KUKA KRL program: EPS_2_251546_SANMH1A_A_20251029061754.src

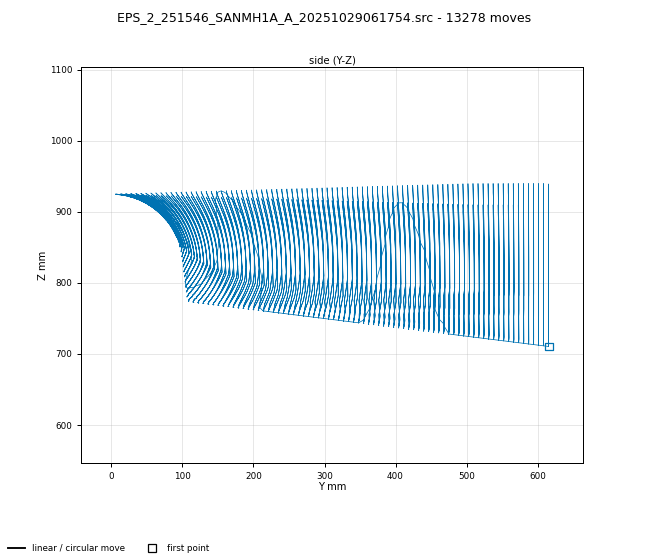
[picture p0: tool path of EPS_2_251546_SANMH1A_A_20251029061754.src, 13278 of 13280 moves have a stored position in this frame; points joined in program order, loops and branches not executed]
&ACCESS RVP
&REL 4
&COMMENT QRS 19112012
&PARAM EDITMASK = *
DEF PART()
EXT BAS (BAS_COMMAND :IN,REAL :IN )
INT I
BAS (#INITMOV,0 )

;KUKA QRS Post kuka4.cps  Date:22-06-2017 !

File_ID=2897

QRS_PRE_INIT()

;Init var - Until changes are made in qrs_pre_init
Outlet_Square_prg=0
Inlet_1_Square_prg=0
Inlet_2_Square_prg=0
Inlet_3_Square_prg=0
Inlet_4_Square_prg=0
Inlet_5_Square_prg=0

Outlet_1={X 0.000, Y 508.730, Z 865.000, B 0.000, E1 0.000 }
Inlet_1={X 0.000, Y 510.870, Z 835.000, B 0.000, E1 180.000 }
Outlet_1_type=150
Inlet_1_type=150
;QRS#1=Sidecore dimensions
;QRS#2=150-6" PVC SDR 28
;QRS#3=150-6" PVC SDR 28
;QRS#4=
;QRS#5=
;QRS#6=
;QRS#7=
;QRS#8=
;QRS#9=10-06 PSX
;QRS#10=10-06 PSX
;QRS#11=
;QRS#12=
;QRS#13=
;QRS#14=
;QRS#15=
;QRS#16=1220x127x1219 4'
;QRS#17=EPS Height
;QRS#18=940
;QRS#19=*
;QRS#20= UPDATED VERSION 22-06-2017
;QRS#21=*
Outlet_Square=070
Inlet_1_Square=070
Inlet_2_Square=0
Inlet_3_Square=0
Inlet_4_Square=0
Inlet_5_Square=0
Mill_Square=1
Outlet_Square_Prg=203
Inlet_1_Square_prg=203

QRS_INIT()

$ADVANCE=5

; T1
PTP {E1 173.424,E2 173.424}
PTP {X 0,Y 615.486,A -85,B 0,C 180,E1 173.424,E2 173.424,E3 0,E4 0,E5 0,E6 0}
QRS_SPEED_INIT()
LIN {X 0,Y 615.486,Z 710.513,A -85,B 0,C 180,E1 173.424,E2 173.424,E3 0,E4 0,E5 0,E6 0} C_VEL
LIN {X 0,Y 615.473,Z 710.502,A -85,B 0,C 180,E1 170.801,E2 170.801} C_VEL
LIN {X 0,Y 615.49,Z 710.493,A -85,B 0,C 180,E1 168.139,E2 168.139} C_VEL
LIN {X 0,Y 615.483,Z 710.506,A -85,B 0,C 180,E1 165.451,E2 165.451} C_VEL
LIN {X 0,Y 615.472,Z 710.505,A -85,B 0,C 180,E1 162.729,E2 162.729} C_VEL
LIN {X 0,Y 615.49,Z 710.493,A -85,B 0,C 180,E1 159.967,E2 159.967} C_VEL
LIN {X 0,Y 615.484,Z 710.511,A -85,B 0,C 180,E1 157.155,E2 157.155} C_VEL
LIN {X 0,Y 615.465,Z 710.503,A -85,B 0,C 180,E1 154.436,E2 154.436} C_VEL
LIN {X 0,Y 615.471,Z 710.498,A -85,B 0,C 180,E1 152.084,E2 152.084} C_VEL
LIN {X 0,Y 615.478,Z 710.496,A -85,B 0,C 180,E1 149.839,E2 149.839} C_VEL
LIN {X 0,Y 615.499,Z 710.493,A -85,B 0,C 180,E1 147.543,E2 147.543} C_VEL
LIN {X 0,Y 615.495,Z 710.499,A -85,B 0,C 180,E1 145.185,E2 145.185} C_VEL
LIN {X 0,Y 615.489,Z 710.514,A -85,B 0,C 180,E1 142.758,E2 142.758} C_VEL
LIN {X 0,Y 615.461,Z 710.501,A -85,B 0,C 180,E1 139.914,E2 139.914} C_VEL
LIN {X 0,Y 615.469,Z 710.497,A -85,B 0,C 180,E1 137.645,E2 137.645} C_VEL
LIN {X 0,Y 615.495,Z 710.5,A -85,B 0,C 180,E1 134.932,E2 134.932} C_VEL
LIN {X 0,Y 615.48,Z 710.511,A -85,B 0,C 180,E1 132.354,E2 132.354} C_VEL
LIN {X 0,Y 615.455,Z 710.503,A -85,B 0,C 180,E1 129.753,E2 129.753} C_VEL
LIN {X 0,Y 615.495,Z 710.497,A -85,B 0,C 180,E1 126.937,E2 126.937} C_VEL
LIN {X 0,Y 615.467,Z 710.508,A -85,B 0,C 180,E1 124.023,E2 124.023} C_VEL
LIN {X 0,Y 615.452,Z 710.505,A -85,B 0,C 180,E1 121.688,E2 121.688} C_VEL
LIN {X 0,Y 615.449,Z 710.503,A -85,B 0,C 180,E1 119.408,E2 119.408} C_VEL
LIN {X 0,Y 615.465,Z 710.499,A -85,B 0,C 180,E1 117.041,E2 117.041} C_VEL
LIN {X 0,Y 615.483,Z 710.511,A -85,B 0,C 180,E1 114.007,E2 114.007} C_VEL
LIN {X 0,Y 615.447,Z 710.505,A -85,B 0,C 180,E1 111.433,E2 111.433} C_VEL
LIN {X 0,Y 615.445,Z 710.505,A -85,B 0,C 180,E1 109.339,E2 109.339} C_VEL
LIN {X 0,Y 615.497,Z 710.635,A -85,B 0,C 180,E1 107.957,E2 107.957} C_VEL
LIN {X 0,Y 615.475,Z 724.409,A -85,B 0,C 180,E1 105.226,E2 105.226} C_VEL
LIN {X 0,Y 615.489,Z 740.007,A -85,B 0,C 180,E1 102.195,E2 102.195} C_VEL
LIN {X 0,Y 615.485,Z 751.04,A -85,B 0,C 180,E1 100.111,E2 100.111} C_VEL
LIN {X 0,Y 615.481,Z 752.153,A -85,B 0,C 180,E1 100.049,E2 100.049} C_VEL
LIN {X 0,Y 615.495,Z 826.708,A -85,B 0,C 180,E1 99.157,E2 99.157} C_VEL
LIN {X 0,Y 615.497,Z 834.892,A -85,B 0,C 180,E1 98.992,E2 98.992} C_VEL
LIN {X 0,Y 615.497,Z 843.45,A -85,B 0,C 180,E1 98.743,E2 98.743} C_VEL
LIN {X 0,Y 615.497,Z 851.061,A -85,B 0,C 180,E1 98.454,E2 98.454} C_VEL
LIN {X 0,Y 615.499,Z 859.582,A -85,B 0,C 180,E1 98.041,E2 98.041} C_VEL
LIN {X 0,Y 615.488,Z 867.749,A -85,B 0,C 180,E1 97.546,E2 97.546} C_VEL
LIN {X 0,Y 615.492,Z 874.389,A -85,B 0,C 180,E1 97.058,E2 97.058} C_VEL
LIN {X 0,Y 615.498,Z 880.184,A -85,B 0,C 180,E1 96.557,E2 96.557} C_VEL
LIN {X 0,Y 615.499,Z 886.535,A -85,B 0,C 180,E1 95.898,E2 95.898} C_VEL
LIN {X 0,Y 615.495,Z 892.984,A -85,B 0,C 180,E1 95.077,E2 95.077} C_VEL
LIN {X 0,Y 615.491,Z 898.123,A -85,B 0,C 180,E1 94.256,E2 94.256} C_VEL
LIN {X 0,Y 615.493,Z 902.886,A -85,B 0,C 180,E1 93.273,E2 93.273} C_VEL
LIN {X 0,Y 615.493,Z 905.2,A -85,B 0,C 180,E1 92.618,E2 92.618} C_VEL
LIN {X 0,Y 615.499,Z 906.976,A -85,B 0,C 180,E1 91.963,E2 91.963} C_VEL
LIN {X 0,Y 615.492,Z 908.266,A -85,B 0,C 180,E1 91.309,E2 91.309} C_VEL
LIN {X 0,Y 615.491,Z 909.083,A -85,B 0,C 180,E1 90.654,E2 90.654} C_VEL
LIN {X 0,Y 615.492,Z 909.384,A -85,B 0,C 180,E1 90,E2 90} C_VEL
LIN {X 0,Y 615.492,Z 909.125,A -85,B 0,C 180,E1 89.346,E2 89.346} C_VEL
LIN {X 0,Y 615.494,Z 908.393,A -85,B 0,C 180,E1 88.691,E2 88.691} C_VEL
LIN {X 0,Y 615.499,Z 907.194,A -85,B 0,C 180,E1 88.037,E2 88.037} C_VEL
LIN {X 0,Y 615.49,Z 904.376,A -85,B 0,C 180,E1 87.055,E2 87.055} C_VEL
LIN {X 0,Y 615.491,Z 901.81,A -85,B 0,C 180,E1 86.399,E2 86.399} C_VEL
LIN {X 0,Y 615.495,Z 896.743,A -85,B 0,C 180,E1 85.416,E2 85.416} C_VEL
LIN {X 0,Y 615.496,Z 891.288,A -85,B 0,C 180,E1 84.595,E2 84.595} C_VEL
LIN {X 0,Y 615.499,Z 884.452,A -85,B 0,C 180,E1 83.773,E2 83.773} C_VEL
LIN {X 0,Y 615.497,Z 877.419,A -85,B 0,C 180,E1 83.1,E2 83.1} C_VEL
LIN {X 0,Y 615.485,Z 869.071,A -85,B 0,C 180,E1 82.454,E2 82.454} C_VEL
LIN {X 0,Y 615.499,Z 861.194,A -85,B 0,C 180,E1 81.959,E2 81.959} C_VEL
LIN {X 0,Y 615.497,Z 853.071,A -85,B 0,C 180,E1 81.546,E2 81.546} C_VEL
LIN {X 0,Y 615.497,Z 844.859,A -85,B 0,C 180,E1 81.215,E2 81.215} C_VEL
LIN {X 0,Y 615.497,Z 836.834,A -85,B 0,C 180,E1 80.967,E2 80.967} C_VEL
LIN {X 0,Y 615.498,Z 827.153,A -85,B 0,C 180,E1 80.76,E2 80.76} C_VEL
LIN {X 0,Y 615.489,Z 751.762,A -85,B 0,C 180,E1 79.847,E2 79.847} C_VEL
LIN {X 0,Y 615.486,Z 750.478,A -85,B 0,C 180,E1 79.722,E2 79.722} C_VEL
LIN {X 0,Y 615.491,Z 735.264,A -85,B 0,C 180,E1 76.799,E2 76.799} C_VEL
LIN {X 0,Y 615.458,Z 721.41,A -85,B 0,C 180,E1 74.094,E2 74.094} C_VEL
LIN {X 0,Y 615.495,Z 710.569,A -85,B 0,C 180,E1 71.922,E2 71.922} C_VEL
LIN {X 0,Y 615.475,Z 710.5,A -85,B 0,C 180,E1 69.269,E2 69.269} C_VEL
LIN {X 0,Y 615.469,Z 710.5,A -85,B 0,C 180,E1 67.155,E2 67.155} C_VEL
LIN {X 0,Y 615.464,Z 710.5,A -85,B 0,C 180,E1 65.007,E2 65.007} C_VEL
LIN {X 0,Y 615.452,Z 710.502,A -85,B 0,C 180,E1 62.821,E2 62.821} C_VEL
LIN {X 0,Y 615.444,Z 710.503,A -85,B 0,C 180,E1 60.591,E2 60.591} C_VEL
LIN {X 0,Y 615.444,Z 710.506,A -85,B 0,C 180,E1 58.312,E2 58.312} C_VEL
LIN {X 0,Y 615.457,Z 710.508,A -85,B 0,C 180,E1 55.976,E2 55.976} C_VEL
LIN {X 0,Y 615.495,Z 710.498,A -85,B 0,C 180,E1 53.063,E2 53.063} C_VEL
LIN {X 0,Y 615.451,Z 710.503,A -85,B 0,C 180,E1 50.247,E2 50.247} C_VEL
LIN {X 0,Y 615.474,Z 710.51,A -85,B 0,C 180,E1 47.646,E2 47.646} C_VEL
LIN {X 0,Y 615.497,Z 710.498,A -85,B 0,C 180,E1 44.932,E2 44.932} C_VEL
LIN {X 0,Y 615.467,Z 710.498,A -85,B 0,C 180,E1 42.355,E2 42.355} C_VEL
LIN {X 0,Y 615.459,Z 710.506,A -85,B 0,C 180,E1 39.752,E2 39.752} C_VEL
LIN {X 0,Y 615.492,Z 710.504,A -85,B 0,C 180,E1 36.937,E2 36.937} C_VEL
LIN {X 0,Y 615.464,Z 710.499,A -85,B 0,C 180,E1 34.024,E2 34.024} C_VEL
LIN {X 0,Y 615.46,Z 710.503,A -85,B 0,C 180,E1 31.687,E2 31.687} C_VEL
LIN {X 0,Y 615.469,Z 710.507,A -85,B 0,C 180,E1 29.407,E2 29.407} C_VEL
LIN {X 0,Y 615.494,Z 710.496,A -85,B 0,C 180,E1 26.444,E2 26.444} C_VEL
LIN {X 0,Y 615.484,Z 710.494,A -85,B 0,C 180,E1 24.007,E2 24.007} C_VEL
LIN {X 0,Y 615.465,Z 710.503,A -85,B 0,C 180,E1 21.433,E2 21.433} C_VEL
LIN {X 0,Y 615.489,Z 710.506,A -85,B 0,C 180,E1 18.605,E2 18.605} C_VEL
LIN {X 0,Y 615.488,Z 710.494,A -85,B 0,C 180,E1 15.905,E2 15.905} C_VEL
LIN {X 0,Y 615.47,Z 710.504,A -85,B 0,C 180,E1 13.202,E2 13.202} C_VEL
LIN {X 0,Y 615.486,Z 710.51,A -85,B 0,C 180,E1 10.527,E2 10.527} C_VEL
LIN {X 0,Y 615.495,Z 710.493,A -85,B 0,C 180,E1 7.876,E2 7.876} C_VEL
LIN {X 0,Y 615.474,Z 710.499,A -85,B 0,C 180,E1 5.241,E2 5.241} C_VEL
LIN {X 0,Y 615.491,Z 710.511,A -85,B 0,C 180,E1 2.618,E2 2.618} C_VEL
LIN {X 0,Y 615.486,Z 710.5,A -85,B 0,C 180,E1 0,E2 0} C_VEL
LIN {X 0,Y 615.495,Z 710.492,A -85,B 0,C 180,E1 -2.618,E2 -2.618} C_VEL
LIN {X 0,Y 615.477,Z 710.504,A -85,B 0,C 180,E1 -5.241,E2 -5.241} C_VEL
LIN {X 0,Y 615.485,Z 710.508,A -85,B 0,C 180,E1 -7.876,E2 -7.876} C_VEL
LIN {X 0,Y 615.492,Z 710.493,A -85,B 0,C 180,E1 -10.527,E2 -10.527} C_VEL
LIN {X 0,Y 615.481,Z 710.499,A -85,B 0,C 180,E1 -13.201,E2 -13.201} C_VEL
LIN {X 0,Y 615.483,Z 710.514,A -85,B 0,C 180,E1 -15.905,E2 -15.905} C_VEL
LIN {X 0,Y 615.492,Z 710.494,A -85,B 0,C 180,E1 -18.646,E2 -18.646} C_VEL
LIN {X 0,Y 615.483,Z 710.5,A -85,B 0,C 180,E1 -21.432,E2 -21.432} C_VEL
LIN {X 0,Y 615.485,Z 710.506,A -85,B 0,C 180,E1 -24.272,E2 -24.272} C_VEL
LIN {X 0,Y 615.489,Z 710.493,A -85,B 0,C 180,E1 -27.177,E2 -27.177} C_VEL
LIN {X 0,Y 615.485,Z 710.504,A -85,B 0,C 180,E1 -29.794,E2 -29.794} C_VEL
LIN {X 0,Y 615.479,Z 710.506,A -85,B 0,C 180,E1 -32.458,E2 -32.458} C_VEL
LIN {X 0,Y 615.497,Z 710.495,A -85,B 0,C 180,E1 -34.814,E2 -34.814} C_VEL
LIN {X 0,Y 615.488,Z 710.493,A -85,B 0,C 180,E1 -37.242,E2 -37.242} C_VEL
LIN {X 0,Y 615.489,Z 710.506,A -85,B 0,C 180,E1 -40.089,E2 -40.089} C_VEL
LIN {X 0,Y 615.498,Z 710.513,A -85,B 0,C 180,E1 -42.352,E2 -42.352} C_VEL
LIN {X 0,Y 615.495,Z 710.494,A -85,B 0,C 180,E1 -45.068,E2 -45.068} C_VEL
LIN {X 0,Y 615.495,Z 710.496,A -85,B 0,C 180,E1 -47.919,E2 -47.919} C_VEL
LIN {X 0,Y 615.49,Z 710.505,A -85,B 0,C 180,E1 -50.25,E2 -50.25} C_VEL
LIN {X 0,Y 615.48,Z 710.501,A -85,B 0,C 180,E1 -53.064,E2 -53.064} C_VEL
LIN {X 0,Y 615.49,Z 710.495,A -85,B 0,C 180,E1 -55.299,E2 -55.299} C_VEL
LIN {X 0,Y 615.484,Z 710.494,A -85,B 0,C 180,E1 -57.67,E2 -57.67} C_VEL
LIN {X 0,Y 615.489,Z 710.51,A -85,B 0,C 180,E1 -60.594,E2 -60.594} C_VEL
LIN {X 0,Y 615.475,Z 710.511,A -85,B 0,C 180,E1 -62.957,E2 -62.957} C_VEL
LIN {X 0,Y 615.484,Z 710.494,A -85,B 0,C 180,E1 -65.728,E2 -65.728} C_VEL
LIN {X 0,Y 615.495,Z 710.502,A -85,B 0,C 180,E1 -68.568,E2 -68.568} C_VEL
LIN {X 0,Y 615.498,Z 710.672,A -85,B 0,C 180,E1 -68.963,E2 -68.963} C_VEL
LIN {X 0,Y 615.491,Z 726.63,A -85,B 0,C 180,E1 -71.557,E2 -71.557} C_VEL
LIN {X 0,Y 615.496,Z 744.77,A -85,B 0,C 180,E1 -74.435,E2 -74.435} C_VEL
LIN {X 0,Y 615.478,Z 763.08,A -85,B 0,C 180,E1 -77.302,E2 -77.302} C_VEL
LIN {X 0,Y 615.493,Z 779.482,A -85,B 0,C 180,E1 -79.826,E2 -79.826} C_VEL
LIN {X 0,Y 615.491,Z 780.6,A -85,B 0,C 180,E1 -79.889,E2 -79.889} C_VEL
LIN {X 0,Y 615.499,Z 856.93,A -85,B 0,C 180,E1 -80.801,E2 -80.801} C_VEL
LIN {X 0,Y 615.497,Z 866.69,A -85,B 0,C 180,E1 -81.008,E2 -81.008} C_VEL
LIN {X 0,Y 615.498,Z 877.15,A -85,B 0,C 180,E1 -81.339,E2 -81.339} C_VEL
LIN {X 0,Y 615.497,Z 887.426,A -85,B 0,C 180,E1 -81.794,E2 -81.794} C_VEL
LIN {X 0,Y 615.491,Z 897.198,A -85,B 0,C 180,E1 -82.372,E2 -82.372} C_VEL
LIN {X 0,Y 615.498,Z 904.934,A -85,B 0,C 180,E1 -82.942,E2 -82.942} C_VEL
LIN {X 0,Y 615.498,Z 910.646,A -85,B 0,C 180,E1 -83.443,E2 -83.443} C_VEL
LIN {X 0,Y 615.499,Z 916.921,A -85,B 0,C 180,E1 -84.102,E2 -84.102} C_VEL
LIN {X 0,Y 615.496,Z 922.135,A -85,B 0,C 180,E1 -84.759,E2 -84.759} C_VEL
LIN {X 0,Y 615.495,Z 926.482,A -85,B 0,C 180,E1 -85.416,E2 -85.416} C_VEL
LIN {X 0,Y 615.492,Z 931.603,A -85,B 0,C 180,E1 -86.399,E2 -86.399} C_VEL
LIN {X 0,Y 615.488,Z 934.221,A -85,B 0,C 180,E1 -87.055,E2 -87.055} C_VEL
LIN {X 0,Y 615.495,Z 937.086,A -85,B 0,C 180,E1 -88.037,E2 -88.037} C_VEL
LIN {X 0,Y 615.494,Z 938.33,A -85,B 0,C 180,E1 -88.691,E2 -88.691} C_VEL
LIN {X 0,Y 615.493,Z 939.104,A -85,B 0,C 180,E1 -89.346,E2 -89.346} C_VEL
LIN {X 0,Y 615.491,Z 939.389,A -85,B 0,C 180,E1 -90,E2 -90} C_VEL
LIN {X 0,Y 615.493,Z 939.104,A -85,B 0,C 180,E1 -90.654,E2 -90.654} C_VEL
LIN {X 0,Y 615.494,Z 938.33,A -85,B 0,C 180,E1 -91.309,E2 -91.309} C_VEL
LIN {X 0,Y 615.495,Z 937.086,A -85,B 0,C 180,E1 -91.963,E2 -91.963} C_VEL
LIN {X 0,Y 615.488,Z 934.221,A -85,B 0,C 180,E1 -92.945,E2 -92.945} C_VEL
LIN {X 0,Y 615.492,Z 931.603,A -85,B 0,C 180,E1 -93.601,E2 -93.601} C_VEL
LIN {X 0,Y 615.495,Z 926.482,A -85,B 0,C 180,E1 -94.584,E2 -94.584} C_VEL
LIN {X 0,Y 615.495,Z 920.968,A -85,B 0,C 180,E1 -95.405,E2 -95.405} C_VEL
LIN {X 0,Y 615.498,Z 914.018,A -85,B 0,C 180,E1 -96.227,E2 -96.227} C_VEL
LIN {X 0,Y 615.497,Z 906.858,A -85,B 0,C 180,E1 -96.901,E2 -96.901} C_VEL
LIN {X 0,Y 615.488,Z 899.621,A -85,B 0,C 180,E1 -97.463,E2 -97.463} C_VEL
LIN {X 0,Y 615.497,Z 891.868,A -85,B 0,C 180,E1 -97.958,E2 -97.958} C_VEL
LIN {X 0,Y 615.498,Z 883.913,A -85,B 0,C 180,E1 -98.371,E2 -98.371} C_VEL
LIN {X 0,Y 615.497,Z 874.754,A -85,B 0,C 180,E1 -98.743,E2 -98.743} C_VEL
LIN {X 0,Y 615.497,Z 866.69,A -85,B 0,C 180,E1 -98.992,E2 -98.992} C_VEL
LIN {X 0,Y 615.499,Z 856.93,A -85,B 0,C 180,E1 -99.199,E2 -99.199} C_VEL
LIN {X 0,Y 615.491,Z 780.6,A -85,B 0,C 180,E1 -100.111,E2 -100.111} C_VEL
LIN {X 0,Y 615.493,Z 779.29,A -85,B 0,C 180,E1 -100.194,E2 -100.194} C_VEL
LIN {X 0,Y 615.479,Z 762.006,A -85,B 0,C 180,E1 -102.866,E2 -102.866} C_VEL
LIN {X 0,Y 615.497,Z 743.691,A -85,B 0,C 180,E1 -105.735,E2 -105.735} C_VEL
LIN {X 0,Y 615.49,Z 725.613,A -85,B 0,C 180,E1 -108.606,E2 -108.606} C_VEL
LIN {X 0,Y 615.498,Z 710.672,A -85,B 0,C 180,E1 -111.037,E2 -111.037} C_VEL
LIN {X 0,Y 615.491,Z 710.501,A -85,B 0,C 180,E1 -113.556,E2 -113.556} C_VEL
LIN {X 0,Y 615.486,Z 710.495,A -85,B 0,C 180,E1 -116.444,E2 -116.444} C_VEL
LIN {X 0,Y 615.485,Z 710.497,A -85,B 0,C 180,E1 -118.658,E2 -118.658} C_VEL
LIN {X 0,Y 615.485,Z 710.507,A -85,B 0,C 180,E1 -121.086,E2 -121.086} C_VEL
LIN {X 0,Y 615.492,Z 710.495,A -85,B 0,C 180,E1 -124.022,E2 -124.022} C_VEL
LIN {X 0,Y 615.484,Z 710.494,A -85,B 0,C 180,E1 -126.425,E2 -126.425} C_VEL
LIN {X 0,Y 615.481,Z 710.503,A -85,B 0,C 180,E1 -129.061,E2 -129.061} C_VEL
LIN {X 0,Y 615.49,Z 710.513,A -85,B 0,C 180,E1 -131.474,E2 -131.474} C_VEL
LIN {X 0,Y 615.496,Z 710.496,A -85,B 0,C 180,E1 -134.149,E2 -134.149} C_VEL
LIN {X 0,Y 615.492,Z 710.495,A -85,B 0,C 180,E1 -136.952,E2 -136.952} C_VEL
LIN {X 0,Y 615.482,Z 710.506,A -85,B 0,C 180,E1 -139.393,E2 -139.393} C_VEL
LIN {X 0,Y 615.489,Z 710.506,A -85,B 0,C 180,E1 -141.988,E2 -141.988} C_VEL
LIN {X 0,Y 615.493,Z 710.496,A -85,B 0,C 180,E1 -144.385,E2 -144.385} C_VEL
LIN {X 0,Y 615.491,Z 710.493,A -85,B 0,C 180,E1 -146.764,E2 -146.764} C_VEL
LIN {X 0,Y 615.49,Z 710.494,A -85,B 0,C 180,E1 -149.08,E2 -149.08} C_VEL
LIN {X 0,Y 615.478,Z 710.504,A -85,B 0,C 180,E1 -151.552,E2 -151.552} C_VEL
LIN {X 0,Y 615.482,Z 710.506,A -85,B 0,C 180,E1 -154.284,E2 -154.284} C_VEL
LIN {X 0,Y 615.49,Z 710.493,A -85,B 0,C 180,E1 -157.156,E2 -157.156} C_VEL
LIN {X 0,Y 615.482,Z 710.511,A -85,B 0,C 180,E1 -159.967,E2 -159.967} C_VEL
LIN {X 0,Y 615.484,Z 710.498,A -85,B 0,C 180,E1 -162.729,E2 -162.729} C_VEL
LIN {X 0,Y 615.492,Z 710.493,A -85,B 0,C 180,E1 -165.451,E2 -165.451} C_VEL
LIN {X 0,Y 615.484,Z 710.511,A -85,B 0,C 180,E1 -168.139,E2 -168.139} C_VEL
LIN {X 0,Y 615.48,Z 710.501,A -85,B 0,C 180,E1 -170.801,E2 -170.801} C_VEL
LIN {X 0,Y 615.492,Z 710.492,A -85,B 0,C 180,E1 -173.443,E2 -173.443} C_VEL
LIN {X 0,Y 615.49,Z 710.502,A -85,B 0,C 180,E1 -176.072,E2 -176.072} C_VEL
LIN {X 0,Y 615.485,Z 710.508,A -85,B 0,C 180,E1 -178.691,E2 -178.691} C_VEL
LIN {X 0,Y 615.483,Z 710.496,A -85,B 0,C 180,E1 -181.309,E2 -181.309} C_VEL
LIN {X 0,Y 615.495,Z 710.494,A -85,B 0,C 180,E1 -183.929,E2 -183.929} C_VEL
LIN {X 0,Y 615.486,Z 710.513,A -85,B 0,C 180,E1 -186.576,E2 -186.576} C_VEL
LIN {X 0,Y 614.801,Z 710.649,A -85,B 0,C 180,E1 -187.122,E2 -187.122} C_VEL
LIN {X 0,Y 611.958,Z 711.063,A -85,B 0,C 180,E1 -188.008,E2 -188.008} C_VEL
LIN {X 0,Y 609.568,Z 711.374,A -85,B 0,C 180,E1 -188.721,E2 -188.721} C_VEL
LIN {X 0,Y 608.541,Z 711.491,A -85,B 0,C 180,E1 -189.27,E2 -189.27} C_VEL
LIN {X 0,Y 608.455,Z 711.499,A -85,B 0,C 180,E1 -189.456,E2 -189.456} C_VEL
LIN {X 0,Y 608.465,Z 711.498,A -85,B 0,C 180,E1 -192,E2 -192} C_VEL
LIN {X 0,Y 608.47,Z 711.507,A -85,B 0,C 180,E1 -194.721,E2 -194.721} C_VEL
LIN {X 0,Y 608.446,Z 711.501,A -85,B 0,C 180,E1 -197.477,E2 -197.477} C_VEL
LIN {X 0,Y 608.468,Z 711.498,A -85,B 0,C 180,E1 -200.274,E2 -200.274} C_VEL
LIN {X 0,Y 608.443,Z 711.509,A -85,B 0,C 180,E1 -203.124,E2 -203.124} C_VEL
LIN {X 0,Y 608.455,Z 711.5,A -85,B 0,C 180,E1 -205.717,E2 -205.717} C_VEL
LIN {X 0,Y 608.453,Z 711.499,A -85,B 0,C 180,E1 -208.267,E2 -208.267} C_VEL
LIN {X 0,Y 608.468,Z 711.499,A -85,B 0,C 180,E1 -210.545,E2 -210.545} C_VEL
LIN {X 0,Y 608.461,Z 711.504,A -85,B 0,C 180,E1 -212.879,E2 -212.879} C_VEL
LIN {X 0,Y 608.438,Z 711.512,A -85,B 0,C 180,E1 -215.278,E2 -215.278} C_VEL
LIN {X 0,Y 608.456,Z 711.502,A -85,B 0,C 180,E1 -217.747,E2 -217.747} C_VEL
LIN {X 0,Y 608.439,Z 711.5,A -85,B 0,C 180,E1 -220.327,E2 -220.327} C_VEL
LIN {X 0,Y 608.48,Z 711.505,A -85,B 0,C 180,E1 -223.31,E2 -223.31} C_VEL
LIN {X 0,Y 608.451,Z 711.5,A -85,B 0,C 180,E1 -226.129,E2 -226.129} C_VEL
LIN {X 0,Y 608.455,Z 711.5,A -85,B 0,C 180,E1 -228.823,E2 -228.823} C_VEL
LIN {X 0,Y 608.454,Z 711.506,A -85,B 0,C 180,E1 -231.761,E2 -231.761} C_VEL
LIN {X 0,Y 608.439,Z 711.506,A -85,B 0,C 180,E1 -233.956,E2 -233.956} C_VEL
LIN {X 0,Y 608.444,Z 711.501,A -85,B 0,C 180,E1 -236.328,E2 -236.328} C_VEL
LIN {X 0,Y 608.442,Z 711.5,A -85,B 0,C 180,E1 -238.733,E2 -238.733} C_VEL
LIN {X 0,Y 608.481,Z 711.5,A -85,B 0,C 180,E1 -241.379,E2 -241.379} C_VEL
LIN {X 0,Y 608.445,Z 711.503,A -85,B 0,C 180,E1 -244.285,E2 -244.285} C_VEL
LIN {X 0,Y 608.429,Z 711.502,A -85,B 0,C 180,E1 -246.875,E2 -246.875} C_VEL
LIN {X 0,Y 608.465,Z 711.505,A -85,B 0,C 180,E1 -249.726,E2 -249.726} C_VEL
LIN {X 0,Y 608.493,Z 711.606,A -85,B 0,C 180,E1 -252.004,E2 -252.004} C_VEL
LIN {X 0,Y 608.457,Z 724.582,A -85,B 0,C 180,E1 -254.594,E2 -254.594} C_VEL
LIN {X 0,Y 608.458,Z 738.509,A -85,B 0,C 180,E1 -257.323,E2 -257.323} C_VEL
LIN {X 0,Y 608.466,Z 751.478,A -85,B 0,C 180,E1 -259.792,E2 -259.792} C_VEL
LIN {X 0,Y 608.516,Z 753.832,A -85,B 0,C 180,E1 -259.856,E2 -259.856} C_VEL
LIN {X 0,Y 608.508,Z 827.252,A -85,B 0,C 180,E1 -260.737,E2 -260.737} C_VEL
LIN {X 0,Y 608.512,Z 836.951,A -85,B 0,C 180,E1 -260.946,E2 -260.946} C_VEL
LIN {X 0,Y 608.499,Z 848.538,A -85,B 0,C 180,E1 -261.323,E2 -261.323} C_VEL
LIN {X 0,Y 608.479,Z 858.432,A -85,B 0,C 180,E1 -261.782,E2 -261.782} C_VEL
LIN {X 0,Y 608.471,Z 866.885,A -85,B 0,C 180,E1 -262.283,E2 -262.283} C_VEL
LIN {X 0,Y 608.46,Z 874.854,A -85,B 0,C 180,E1 -262.867,E2 -262.867} C_VEL
LIN {X 0,Y 608.467,Z 881.903,A -85,B 0,C 180,E1 -263.496,E2 -263.496} C_VEL
LIN {X 0,Y 608.458,Z 888.396,A -85,B 0,C 180,E1 -264.199,E2 -264.199} C_VEL
LIN {X 0,Y 608.437,Z 894.642,A -85,B 0,C 180,E1 -265.03,E2 -265.03} C_VEL
LIN {X 0,Y 608.432,Z 900.425,A -85,B 0,C 180,E1 -266.026,E2 -266.026} C_VEL
LIN {X 0,Y 608.447,Z 904.63,A -85,B 0,C 180,E1 -267.021,E2 -267.021} C_VEL
LIN {X 0,Y 608.443,Z 907.569,A -85,B 0,C 180,E1 -268.014,E2 -268.014} C_VEL
LIN {X 0,Y 608.445,Z 908.87,A -85,B 0,C 180,E1 -268.676,E2 -268.676} C_VEL
LIN {X 0,Y 608.434,Z 909.692,A -85,B 0,C 180,E1 -269.338,E2 -269.338} C_VEL
LIN {X 0,Y 608.432,Z 909.995,A -85,B 0,C 180,E1 -270,E2 -270} C_VEL
LIN {X 0,Y 608.435,Z 909.735,A -85,B 0,C 180,E1 -270.662,E2 -270.662} C_VEL
LIN {X 0,Y 608.446,Z 908.997,A -85,B 0,C 180,E1 -271.324,E2 -271.324} C_VEL
LIN {X 0,Y 608.444,Z 907.787,A -85,B 0,C 180,E1 -271.986,E2 -271.986} C_VEL
LIN {X 0,Y 608.445,Z 904.941,A -85,B 0,C 180,E1 -272.979,E2 -272.979} C_VEL
LIN {X 0,Y 608.445,Z 902.352,A -85,B 0,C 180,E1 -273.642,E2 -273.642} C_VEL
LIN {X 0,Y 608.445,Z 897.244,A -85,B 0,C 180,E1 -274.638,E2 -274.638} C_VEL
LIN {X 0,Y 608.461,Z 891.748,A -85,B 0,C 180,E1 -275.468,E2 -275.468} C_VEL
LIN {X 0,Y 608.455,Z 884.144,A -85,B 0,C 180,E1 -276.374,E2 -276.374} C_VEL
LIN {X 0,Y 608.463,Z 875.948,A -85,B 0,C 180,E1 -277.133,E2 -277.133} C_VEL
LIN {X 0,Y 608.467,Z 868.198,A -85,B 0,C 180,E1 -277.717,E2 -277.717} C_VEL
LIN {X 0,Y 608.48,Z 860.032,A -85,B 0,C 180,E1 -278.218,E2 -278.218} C_VEL
LIN {X 0,Y 608.484,Z 849.674,A -85,B 0,C 180,E1 -278.719,E2 -278.719} C_VEL
LIN {X 0,Y 608.51,Z 838.029,A -85,B 0,C 180,E1 -279.117,E2 -279.117} C_VEL
LIN {X 0,Y 608.517,Z 827.635,A -85,B 0,C 180,E1 -279.347,E2 -279.347} C_VEL
LIN {X 0,Y 608.509,Z 781.173,A -85,B 0,C 180,E1 -279.913,E2 -279.913} C_VEL
LIN {X 0,Y 608.484,Z 751.922,A -85,B 0,C 180,E1 -280.271,E2 -280.271} C_VEL
LIN {X 0,Y 608.457,Z 750.745,A -85,B 0,C 180,E1 -280.398,E2 -280.398} C_VEL
LIN {X 0,Y 608.463,Z 735.488,A -85,B 0,C 180,E1 -283.356,E2 -283.356} C_VEL
LIN {X 0,Y 608.452,Z 721.556,A -85,B 0,C 180,E1 -286.094,E2 -286.094} C_VEL
LIN {X 0,Y 608.471,Z 711.572,A -85,B 0,C 180,E1 -288.106,E2 -288.106} C_VEL
LIN {X 0,Y 608.438,Z 711.501,A -85,B 0,C 180,E1 -290.982,E2 -290.982} C_VEL
LIN {X 0,Y 608.425,Z 711.503,A -85,B 0,C 180,E1 -293.125,E2 -293.125} C_VEL
LIN {X 0,Y 608.439,Z 711.503,A -85,B 0,C 180,E1 -295.714,E2 -295.714} C_VEL
LIN {X 0,Y 608.482,Z 711.501,A -85,B 0,C 180,E1 -298.621,E2 -298.621} C_VEL
LIN {X 0,Y 608.437,Z 711.501,A -85,B 0,C 180,E1 -301.318,E2 -301.318} C_VEL
LIN {X 0,Y 608.425,Z 711.504,A -85,B 0,C 180,E1 -303.728,E2 -303.728} C_VEL
LIN {X 0,Y 608.439,Z 711.506,A -85,B 0,C 180,E1 -306.093,E2 -306.093} C_VEL
LIN {X 0,Y 608.467,Z 711.507,A -85,B 0,C 180,E1 -308.588,E2 -308.588} C_VEL
LIN {X 0,Y 608.452,Z 711.5,A -85,B 0,C 180,E1 -311.341,E2 -311.341} C_VEL
LIN {X 0,Y 608.446,Z 711.501,A -85,B 0,C 180,E1 -313.872,E2 -313.872} C_VEL
LIN {X 0,Y 608.48,Z 711.506,A -85,B 0,C 180,E1 -316.69,E2 -316.69} C_VEL
LIN {X 0,Y 608.454,Z 711.499,A -85,B 0,C 180,E1 -319.697,E2 -319.697} C_VEL
LIN {X 0,Y 608.481,Z 711.506,A -85,B 0,C 180,E1 -322.84,E2 -322.84} C_VEL
LIN {X 0,Y 608.469,Z 711.498,A -85,B 0,C 180,E1 -325.531,E2 -325.531} C_VEL
LIN {X 0,Y 608.462,Z 711.498,A -85,B 0,C 180,E1 -327.905,E2 -327.905} C_VEL
LIN {X 0,Y 608.448,Z 711.5,A -85,B 0,C 180,E1 -330.219,E2 -330.219} C_VEL
LIN {X 0,Y 608.479,Z 711.503,A -85,B 0,C 180,E1 -332.793,E2 -332.793} C_VEL
LIN {X 0,Y 608.48,Z 711.496,A -85,B 0,C 180,E1 -335.847,E2 -335.847} C_VEL
LIN {X 0,Y 608.461,Z 711.498,A -85,B 0,C 180,E1 -338.308,E2 -338.308} C_VEL
LIN {X 0,Y 608.454,Z 711.51,A -85,B 0,C 180,E1 -341.13,E2 -341.13} C_VEL
LIN {X 0,Y 608.465,Z 711.498,A -85,B 0,C 180,E1 -343.906,E2 -343.906} C_VEL
LIN {X 0,Y 608.454,Z 711.5,A -85,B 0,C 180,E1 -346.643,E2 -346.643} C_VEL
LIN {X 0,Y 608.463,Z 711.509,A -85,B 0,C 180,E1 -349.35,E2 -349.35} C_VEL
LIN {X 0,Y 608.485,Z 711.496,A -85,B 0,C 180,E1 -352.033,E2 -352.033} C_VEL
LIN {X 0,Y 608.456,Z 711.499,A -85,B 0,C 180,E1 -354.698,E2 -354.698} C_VEL
LIN {X 0,Y 608.482,Z 711.505,A -85,B 0,C 180,E1 -357.352,E2 -357.352} C_VEL
LIN {X 0,Y 608.477,Z 711.499,A -85,B 0,C 180,E1 -360,E2 -360} C_VEL
LIN {X 0,Y 608.484,Z 711.495,A -85,B 0,C 180,E1 -362.648,E2 -362.648} C_VEL
LIN {X 0,Y 608.458,Z 711.504,A -85,B 0,C 180,E1 -365.302,E2 -365.302} C_VEL
LIN {X 0,Y 608.479,Z 711.502,A -85,B 0,C 180,E1 -367.967,E2 -367.967} C_VEL
LIN {X 0,Y 608.472,Z 711.497,A -85,B 0,C 180,E1 -370.956,E2 -370.956} C_VEL
LIN {X 0,Y 608.462,Z 711.501,A -85,B 0,C 180,E1 -373.356,E2 -373.356} C_VEL
LIN {X 0,Y 608.462,Z 711.505,A -85,B 0,C 180,E1 -376.094,E2 -376.094} C_VEL
LIN {X 0,Y 608.459,Z 711.498,A -85,B 0,C 180,E1 -378.869,E2 -378.869} C_VEL
LIN {X 0,Y 608.467,Z 711.503,A -85,B 0,C 180,E1 -381.692,E2 -381.692} C_VEL
LIN {X 0,Y 608.455,Z 711.501,A -85,B 0,C 180,E1 -384.571,E2 -384.571} C_VEL
LIN {X 0,Y 608.483,Z 711.495,A -85,B 0,C 180,E1 -387.208,E2 -387.208} C_VEL
LIN {X 0,Y 608.469,Z 711.505,A -85,B 0,C 180,E1 -389.971,E2 -389.971} C_VEL
LIN {X 0,Y 608.456,Z 711.504,A -85,B 0,C 180,E1 -392.521,E2 -392.521} C_VEL
LIN {X 0,Y 608.452,Z 711.499,A -85,B 0,C 180,E1 -395.277,E2 -395.277} C_VEL
LIN {X 0,Y 608.472,Z 711.499,A -85,B 0,C 180,E1 -397.746,E2 -397.746} C_VEL
LIN {X 0,Y 608.452,Z 711.51,A -85,B 0,C 180,E1 -400.329,E2 -400.329} C_VEL
LIN {X 0,Y 608.46,Z 711.5,A -85,B 0,C 180,E1 -402.959,E2 -402.959} C_VEL
LIN {X 0,Y 608.464,Z 711.499,A -85,B 0,C 180,E1 -405.735,E2 -405.735} C_VEL
LIN {X 0,Y 608.465,Z 711.506,A -85,B 0,C 180,E1 -408.657,E2 -408.657} C_VEL
LIN {X 0,Y 608.472,Z 711.497,A -85,B 0,C 180,E1 -411.412,E2 -411.412} C_VEL
LIN {X 0,Y 608.48,Z 711.497,A -85,B 0,C 180,E1 -413.95,E2 -413.95} C_VEL
LIN {X 0,Y 608.469,Z 711.503,A -85,B 0,C 180,E1 -416.33,E2 -416.33} C_VEL
LIN {X 0,Y 608.479,Z 711.507,A -85,B 0,C 180,E1 -418.727,E2 -418.727} C_VEL
LIN {X 0,Y 608.473,Z 711.498,A -85,B 0,C 180,E1 -421.38,E2 -421.38} C_VEL
LIN {X 0,Y 608.481,Z 711.498,A -85,B 0,C 180,E1 -424.277,E2 -424.277} C_VEL
LIN {X 0,Y 608.45,Z 711.511,A -85,B 0,C 180,E1 -426.876,E2 -426.876} C_VEL
LIN {X 0,Y 608.489,Z 711.683,A -85,B 0,C 180,E1 -428.887,E2 -428.887} C_VEL
LIN {X 0,Y 608.514,Z 726.278,A -85,B 0,C 180,E1 -431.272,E2 -431.272} C_VEL
LIN {X 0,Y 608.503,Z 744.878,A -85,B 0,C 180,E1 -434.251,E2 -434.251} C_VEL
LIN {X 0,Y 608.452,Z 763.263,A -85,B 0,C 180,E1 -437.153,E2 -437.153} C_VEL
LIN {X 0,Y 608.47,Z 779.912,A -85,B 0,C 180,E1 -439.729,E2 -439.729} C_VEL
LIN {X 0,Y 608.52,Z 782.297,A -85,B 0,C 180,E1 -439.793,E2 -439.793} C_VEL
LIN {X 0,Y 608.504,Z 856.143,A -85,B 0,C 180,E1 -440.674,E2 -440.674} C_VEL
LIN {X 0,Y 608.496,Z 865.413,A -85,B 0,C 180,E1 -440.862,E2 -440.862} C_VEL
LIN {X 0,Y 608.489,Z 873.887,A -85,B 0,C 180,E1 -441.113,E2 -441.113} C_VEL
LIN {X 0,Y 608.501,Z 882.387,A -85,B 0,C 180,E1 -441.448,E2 -441.448} C_VEL
LIN {X 0,Y 608.497,Z 890.718,A -85,B 0,C 180,E1 -441.866,E2 -441.866} C_VEL
LIN {X 0,Y 608.469,Z 898.759,A -85,B 0,C 180,E1 -442.367,E2 -442.367} C_VEL
LIN {X 0,Y 608.484,Z 906.414,A -85,B 0,C 180,E1 -442.951,E2 -442.951} C_VEL
LIN {X 0,Y 608.452,Z 914.437,A -85,B 0,C 180,E1 -443.7,E2 -443.7} C_VEL
LIN {X 0,Y 608.46,Z 921.43,A -85,B 0,C 180,E1 -444.532,E2 -444.532} C_VEL
LIN {X 0,Y 608.431,Z 926.985,A -85,B 0,C 180,E1 -445.362,E2 -445.362} C_VEL
LIN {X 0,Y 608.446,Z 932.146,A -85,B 0,C 180,E1 -446.358,E2 -446.358} C_VEL
LIN {X 0,Y 608.444,Z 934.786,A -85,B 0,C 180,E1 -447.021,E2 -447.021} C_VEL
LIN {X 0,Y 608.44,Z 937.678,A -85,B 0,C 180,E1 -448.014,E2 -448.014} C_VEL
LIN {X 0,Y 608.446,Z 938.934,A -85,B 0,C 180,E1 -448.676,E2 -448.676} C_VEL
LIN {X 0,Y 608.436,Z 939.714,A -85,B 0,C 180,E1 -449.338,E2 -449.338} C_VEL
LIN {X 0,Y 608.431,Z 940,A -85,B 0,C 180,E1 -450,E2 -450} C_VEL
LIN {X 0,Y 608.436,Z 939.714,A -85,B 0,C 180,E1 -450.662,E2 -450.662} C_VEL
LIN {X 0,Y 608.446,Z 938.933,A -85,B 0,C 180,E1 -451.324,E2 -451.324} C_VEL
LIN {X 0,Y 608.44,Z 937.678,A -85,B 0,C 180,E1 -451.986,E2 -451.986} C_VEL
LIN {X 0,Y 608.444,Z 934.786,A -85,B 0,C 180,E1 -452.979,E2 -452.979} C_VEL
LIN {X 0,Y 608.446,Z 932.146,A -85,B 0,C 180,E1 -453.642,E2 -453.642} C_VEL
LIN {X 0,Y 608.431,Z 926.985,A -85,B 0,C 180,E1 -454.638,E2 -454.638} C_VEL
LIN {X 0,Y 608.46,Z 921.429,A -85,B 0,C 180,E1 -455.468,E2 -455.468} C_VEL
LIN {X 0,Y 608.455,Z 913.67,A -85,B 0,C 180,E1 -456.376,E2 -456.376} C_VEL
LIN {X 0,Y 608.484,Z 906.414,A -85,B 0,C 180,E1 -457.049,E2 -457.049} C_VEL
LIN {X 0,Y 608.469,Z 898.759,A -85,B 0,C 180,E1 -457.633,E2 -457.633} C_VEL
LIN {X 0,Y 608.497,Z 890.718,A -85,B 0,C 180,E1 -458.134,E2 -458.134} C_VEL
LIN {X 0,Y 608.501,Z 882.387,A -85,B 0,C 180,E1 -458.552,E2 -458.552} C_VEL
LIN {X 0,Y 608.489,Z 873.887,A -85,B 0,C 180,E1 -458.887,E2 -458.887} C_VEL
LIN {X 0,Y 608.517,Z 864.583,A -85,B 0,C 180,E1 -459.158,E2 -459.158} C_VEL
LIN {X 0,Y 608.518,Z 854.845,A -85,B 0,C 180,E1 -459.347,E2 -459.347} C_VEL
LIN {X 0,Y 608.48,Z 780.236,A -85,B 0,C 180,E1 -460.25,E2 -460.25} C_VEL
LIN {X 0,Y 608.444,Z 777.321,A -85,B 0,C 180,E1 -460.65,E2 -460.65} C_VEL
LIN {X 0,Y 608.476,Z 760.018,A -85,B 0,C 180,E1 -463.356,E2 -463.356} C_VEL
LIN {X 0,Y 608.504,Z 741.677,A -85,B 0,C 180,E1 -466.258,E2 -466.258} C_VEL
LIN {X 0,Y 608.496,Z 724.331,A -85,B 0,C 180,E1 -469.043,E2 -469.043} C_VEL
LIN {X 0,Y 608.475,Z 711.621,A -85,B 0,C 180,E1 -471.136,E2 -471.136} C_VEL
LIN {X 0,Y 608.466,Z 711.498,A -85,B 0,C 180,E1 -473.845,E2 -473.845} C_VEL
LIN {X 0,Y 608.453,Z 711.499,A -85,B 0,C 180,E1 -476.035,E2 -476.035} C_VEL
LIN {X 0,Y 608.473,Z 711.498,A -85,B 0,C 180,E1 -478.62,E2 -478.62} C_VEL
LIN {X 0,Y 608.478,Z 711.507,A -85,B 0,C 180,E1 -481.316,E2 -481.316} C_VEL
LIN {X 0,Y 608.478,Z 711.501,A -85,B 0,C 180,E1 -483.736,E2 -483.736} C_VEL
LIN {X 0,Y 608.479,Z 711.497,A -85,B 0,C 180,E1 -486.09,E2 -486.09} C_VEL
LIN {X 0,Y 608.472,Z 711.497,A -85,B 0,C 180,E1 -488.588,E2 -488.588} C_VEL
LIN {X 0,Y 608.464,Z 711.505,A -85,B 0,C 180,E1 -491.342,E2 -491.342} C_VEL
LIN {X 0,Y 608.464,Z 711.499,A -85,B 0,C 180,E1 -494.265,E2 -494.265} C_VEL
LIN {X 0,Y 608.46,Z 711.5,A -85,B 0,C 180,E1 -497.041,E2 -497.041} C_VEL
LIN {X 0,Y 608.453,Z 711.51,A -85,B 0,C 180,E1 -499.697,E2 -499.697} C_VEL
LIN {X 0,Y 608.472,Z 711.499,A -85,B 0,C 180,E1 -502.254,E2 -502.254} C_VEL
LIN {X 0,Y 608.487,Z 711.496,A -85,B 0,C 180,E1 -505.09,E2 -505.09} C_VEL
LIN {X 0,Y 608.464,Z 711.508,A -85,B 0,C 180,E1 -507.906,E2 -507.906} C_VEL
LIN {X 0,Y 608.471,Z 711.502,A -85,B 0,C 180,E1 -510.221,E2 -510.221} C_VEL
LIN {X 0,Y 608.483,Z 711.496,A -85,B 0,C 180,E1 -512.792,E2 -512.792} C_VEL
LIN {X 0,Y 608.454,Z 711.501,A -85,B 0,C 180,E1 -515.429,E2 -515.429} C_VEL
LIN {X 0,Y 608.466,Z 711.504,A -85,B 0,C 180,E1 -518.308,E2 -518.308} C_VEL
LIN {X 0,Y 608.476,Z 711.496,A -85,B 0,C 180,E1 -521.283,E2 -521.283} C_VEL
LIN {X 0,Y 608.463,Z 711.504,A -85,B 0,C 180,E1 -523.906,E2 -523.906} C_VEL
LIN {X 0,Y 608.462,Z 711.502,A -85,B 0,C 180,E1 -526.644,E2 -526.644} C_VEL
LIN {X 0,Y 608.47,Z 711.497,A -85,B 0,C 180,E1 -529.35,E2 -529.35} C_VEL
LIN {X 0,Y 608.477,Z 711.501,A -85,B 0,C 180,E1 -532.033,E2 -532.033} C_VEL
LIN {X 0,Y 608.459,Z 711.504,A -85,B 0,C 180,E1 -534.698,E2 -534.698} C_VEL
LIN {X 0,Y 608.485,Z 711.495,A -85,B 0,C 180,E1 -537.352,E2 -537.352} C_VEL
LIN {X 0,Y 608.479,Z 711.498,A -85,B 0,C 180,E1 -540,E2 -540} C_VEL
LIN {X 0,Y 608.485,Z 711.505,A -85,B 0,C 180,E1 -542.648,E2 -542.648} C_VEL
LIN {X 0,Y 608.457,Z 711.499,A -85,B 0,C 180,E1 -545.302,E2 -545.302} C_VEL
LIN {X 0,Y 608.485,Z 711.495,A -85,B 0,C 180,E1 -547.967,E2 -547.967} C_VEL
LIN {X 0,Y 608.455,Z 711.499,A -85,B 0,C 180,E1 -549.456,E2 -549.456} C_VEL
LIN {X 0,Y 607.785,Z 711.584,A -85,B 0,C 180,E1 -550.009,E2 -550.009} C_VEL
LIN {X 0,Y 604.936,Z 711.945,A -85,B 0,C 180,E1 -550.906,E2 -550.906} C_VEL
LIN {X 0,Y 602.53,Z 712.241,A -85,B 0,C 180,E1 -551.627,E2 -551.627} C_VEL
LIN {X 0,Y 601.496,Z 712.368,A -85,B 0,C 180,E1 -552.184,E2 -552.184} C_VEL
LIN {X 0,Y 601.411,Z 712.38,A -85,B 0,C 180,E1 -552.372,E2 -552.372} C_VEL
LIN {X 0,Y 601.425,Z 712.384,A -85,B 0,C 180,E1 -554.897,E2 -554.897} C_VEL
LIN {X 0,Y 601.43,Z 712.382,A -85,B 0,C 180,E1 -556.986,E2 -556.986} C_VEL
LIN {X 0,Y 601.404,Z 712.377,A -85,B 0,C 180,E1 -559.81,E2 -559.81} C_VEL
LIN {X 0,Y 601.418,Z 712.38,A -85,B 0,C 180,E1 -562.606,E2 -562.606} C_VEL
LIN {X 0,Y 601.403,Z 712.386,A -85,B 0,C 180,E1 -564.879,E2 -564.879} C_VEL
LIN {X 0,Y 601.417,Z 712.381,A -85,B 0,C 180,E1 -567.362,E2 -567.362} C_VEL
LIN {X 0,Y 601.41,Z 712.383,A -85,B 0,C 180,E1 -569.394,E2 -569.394} C_VEL
LIN {X 0,Y 601.401,Z 712.379,A -85,B 0,C 180,E1 -571.727,E2 -571.727} C_VEL
LIN {X 0,Y 601.421,Z 712.375,A -85,B 0,C 180,E1 -574.119,E2 -574.119} C_VEL
LIN {X 0,Y 601.437,Z 712.382,A -85,B 0,C 180,E1 -577.382,E2 -577.382} C_VEL
LIN {X 0,Y 601.401,Z 712.378,A -85,B 0,C 180,E1 -579.996,E2 -579.996} C_VEL
LIN {X 0,Y 601.411,Z 712.375,A -85,B 0,C 180,E1 -582.67,E2 -582.67} C_VEL
LIN {X 0,Y 601.4,Z 712.389,A -85,B 0,C 180,E1 -585.479,E2 -585.479} C_VEL
LIN {X 0,Y 601.416,Z 712.376,A -85,B 0,C 180,E1 -588.408,E2 -588.408} C_VEL
LIN {X 0,Y 601.414,Z 712.377,A -85,B 0,C 180,E1 -590.874,E2 -590.874} C_VEL
LIN {X 0,Y 601.407,Z 712.384,A -85,B 0,C 180,E1 -593.417,E2 -593.417} C_VEL
LIN {X 0,Y 601.405,Z 712.381,A -85,B 0,C 180,E1 -596.068,E2 -596.068} C_VEL
LIN {X 0,Y 601.415,Z 712.376,A -85,B 0,C 180,E1 -598.546,E2 -598.546} C_VEL
LIN {X 0,Y 601.439,Z 712.377,A -85,B 0,C 180,E1 -601.373,E2 -601.373} C_VEL
LIN {X 0,Y 601.392,Z 712.384,A -85,B 0,C 180,E1 -604.137,E2 -604.137} C_VEL
LIN {X 0,Y 601.382,Z 712.381,A -85,B 0,C 180,E1 -606.588,E2 -606.588} C_VEL
LIN {X 0,Y 601.433,Z 712.377,A -85,B 0,C 180,E1 -609.478,E2 -609.478} C_VEL
LIN {X 0,Y 601.453,Z 712.477,A -85,B 0,C 180,E1 -611.962,E2 -611.962} C_VEL
LIN {X 0,Y 601.425,Z 726.326,A -85,B 0,C 180,E1 -614.756,E2 -614.756} C_VEL
LIN {X 0,Y 601.384,Z 740.253,A -85,B 0,C 180,E1 -617.514,E2 -617.514} C_VEL
LIN {X 0,Y 601.392,Z 751.487,A -85,B 0,C 180,E1 -619.67,E2 -619.67} C_VEL
LIN {X 0,Y 601.527,Z 753.877,A -85,B 0,C 180,E1 -619.737,E2 -619.737} C_VEL
LIN {X 0,Y 601.524,Z 827.285,A -85,B 0,C 180,E1 -620.628,E2 -620.628} C_VEL
LIN {X 0,Y 601.487,Z 837.805,A -85,B 0,C 180,E1 -620.861,E2 -620.861} C_VEL
LIN {X 0,Y 601.473,Z 849.542,A -85,B 0,C 180,E1 -621.263,E2 -621.263} C_VEL
LIN {X 0,Y 601.455,Z 859.93,A -85,B 0,C 180,E1 -621.77,E2 -621.77} C_VEL
LIN {X 0,Y 601.435,Z 868.113,A -85,B 0,C 180,E1 -622.277,E2 -622.277} C_VEL
LIN {X 0,Y 601.414,Z 875.875,A -85,B 0,C 180,E1 -622.868,E2 -622.868} C_VEL
LIN {X 0,Y 601.394,Z 883.708,A -85,B 0,C 180,E1 -623.598,E2 -623.598} C_VEL
LIN {X 0,Y 601.383,Z 891.115,A -85,B 0,C 180,E1 -624.467,E2 -624.467} C_VEL
LIN {X 0,Y 601.34,Z 896.729,A -85,B 0,C 180,E1 -625.307,E2 -625.307} C_VEL
LIN {X 0,Y 601.365,Z 901.943,A -85,B 0,C 180,E1 -626.315,E2 -626.315} C_VEL
LIN {X 0,Y 601.345,Z 904.633,A -85,B 0,C 180,E1 -626.985,E2 -626.985} C_VEL
LIN {X 0,Y 601.342,Z 907.572,A -85,B 0,C 180,E1 -627.991,E2 -627.991} C_VEL
LIN {X 0,Y 601.345,Z 908.871,A -85,B 0,C 180,E1 -628.661,E2 -628.661} C_VEL
LIN {X 0,Y 601.335,Z 909.692,A -85,B 0,C 180,E1 -629.33,E2 -629.33} C_VEL
LIN {X 0,Y 601.333,Z 909.996,A -85,B 0,C 180,E1 -630,E2 -630} C_VEL
LIN {X 0,Y 601.336,Z 909.734,A -85,B 0,C 180,E1 -630.67,E2 -630.67} C_VEL
LIN {X 0,Y 601.346,Z 908.997,A -85,B 0,C 180,E1 -631.339,E2 -631.339} C_VEL
LIN {X 0,Y 601.343,Z 907.786,A -85,B 0,C 180,E1 -632.009,E2 -632.009} C_VEL
LIN {X 0,Y 601.344,Z 904.94,A -85,B 0,C 180,E1 -633.015,E2 -633.015} C_VEL
LIN {X 0,Y 601.364,Z 902.35,A -85,B 0,C 180,E1 -633.685,E2 -633.685} C_VEL
LIN {X 0,Y 601.362,Z 897.242,A -85,B 0,C 180,E1 -634.692,E2 -634.692} C_VEL
LIN {X 0,Y 601.384,Z 891.745,A -85,B 0,C 180,E1 -635.533,E2 -635.533} C_VEL
LIN {X 0,Y 601.395,Z 883.585,A -85,B 0,C 180,E1 -636.504,E2 -636.504} C_VEL
LIN {X 0,Y 601.413,Z 875.943,A -85,B 0,C 180,E1 -637.217,E2 -637.217} C_VEL
LIN {X 0,Y 601.41,Z 868.193,A -85,B 0,C 180,E1 -637.808,E2 -637.808} C_VEL
LIN {X 0,Y 601.447,Z 860.026,A -85,B 0,C 180,E1 -638.314,E2 -638.314} C_VEL
LIN {X 0,Y 601.461,Z 849.66,A -85,B 0,C 180,E1 -638.822,E2 -638.822} C_VEL
LIN {X 0,Y 601.492,Z 838.01,A -85,B 0,C 180,E1 -639.224,E2 -639.224} C_VEL
LIN {X 0,Y 601.532,Z 827.603,A -85,B 0,C 180,E1 -639.457,E2 -639.457} C_VEL
LIN {X 0,Y 601.541,Z 777.55,A -85,B 0,C 180,E1 -640.072,E2 -640.072} C_VEL
LIN {X 0,Y 601.44,Z 751.898,A -85,B 0,C 180,E1 -640.393,E2 -640.393} C_VEL
LIN {X 0,Y 601.369,Z 750.737,A -85,B 0,C 180,E1 -640.521,E2 -640.521} C_VEL
LIN {X 0,Y 601.4,Z 737.227,A -85,B 0,C 180,E1 -643.172,E2 -643.172} C_VEL
LIN {X 0,Y 601.397,Z 723.294,A -85,B 0,C 180,E1 -645.94,E2 -645.94} C_VEL
LIN {X 0,Y 601.441,Z 712.462,A -85,B 0,C 180,E1 -648.149,E2 -648.149} C_VEL
LIN {X 0,Y 601.39,Z 712.379,A -85,B 0,C 180,E1 -651.24,E2 -651.24} C_VEL
LIN {X 0,Y 601.45,Z 712.381,A -85,B 0,C 180,E1 -654.141,E2 -654.141} C_VEL
LIN {X 0,Y 601.396,Z 712.378,A -85,B 0,C 180,E1 -657.114,E2 -657.114} C_VEL
LIN {X 0,Y 601.398,Z 712.378,A -85,B 0,C 180,E1 -659.394,E2 -659.394} C_VEL
LIN {X 0,Y 601.394,Z 712.379,A -85,B 0,C 180,E1 -661.727,E2 -661.727} C_VEL
LIN {X 0,Y 601.413,Z 712.382,A -85,B 0,C 180,E1 -664.119,E2 -664.119} C_VEL
LIN {X 0,Y 601.434,Z 712.373,A -85,B 0,C 180,E1 -667.382,E2 -667.382} C_VEL
LIN {X 0,Y 601.4,Z 712.38,A -85,B 0,C 180,E1 -669.996,E2 -669.996} C_VEL
LIN {X 0,Y 601.412,Z 712.386,A -85,B 0,C 180,E1 -672.67,E2 -672.67} C_VEL
LIN {X 0,Y 601.4,Z 712.377,A -85,B 0,C 180,E1 -675.479,E2 -675.479} C_VEL
LIN {X 0,Y 601.418,Z 712.379,A -85,B 0,C 180,E1 -678.408,E2 -678.408} C_VEL
LIN {X 0,Y 601.405,Z 712.386,A -85,B 0,C 180,E1 -680.873,E2 -680.873} C_VEL
LIN {X 0,Y 601.405,Z 712.379,A -85,B 0,C 180,E1 -683.417,E2 -683.417} C_VEL
LIN {X 0,Y 601.418,Z 712.376,A -85,B 0,C 180,E1 -686.067,E2 -686.067} C_VEL
LIN {X 0,Y 601.418,Z 712.38,A -85,B 0,C 180,E1 -688.546,E2 -688.546} C_VEL
LIN {X 0,Y 601.438,Z 712.377,A -85,B 0,C 180,E1 -691.373,E2 -691.373} C_VEL
LIN {X 0,Y 601.402,Z 712.378,A -85,B 0,C 180,E1 -693.636,E2 -693.636} C_VEL
LIN {X 0,Y 601.459,Z 712.37,A -85,B 0,C 180,E1 -695.86,E2 -695.86} C_VEL
LIN {X 0,Y 601.405,Z 712.382,A -85,B 0,C 180,E1 -698.761,E2 -698.761} C_VEL
LIN {X 0,Y 601.425,Z 712.377,A -85,B 0,C 180,E1 -701.608,E2 -701.608} C_VEL
LIN {X 0,Y 601.445,Z 712.374,A -85,B 0,C 180,E1 -703.713,E2 -703.713} C_VEL
LIN {X 0,Y 601.413,Z 712.377,A -85,B 0,C 180,E1 -706.484,E2 -706.484} C_VEL
LIN {X 0,Y 601.418,Z 712.385,A -85,B 0,C 180,E1 -709.224,E2 -709.224} C_VEL
LIN {X 0,Y 601.447,Z 712.373,A -85,B 0,C 180,E1 -711.939,E2 -711.939} C_VEL
LIN {X 0,Y 601.423,Z 712.375,A -85,B 0,C 180,E1 -714.636,E2 -714.636} C_VEL
LIN {X 0,Y 601.447,Z 712.38,A -85,B 0,C 180,E1 -717.321,E2 -717.321} C_VEL
LIN {X 0,Y 601.446,Z 712.375,A -85,B 0,C 180,E1 -720,E2 -720} C_VEL
LIN {X 0,Y 601.449,Z 712.371,A -85,B 0,C 180,E1 -722.679,E2 -722.679} C_VEL
LIN {X 0,Y 601.422,Z 712.381,A -85,B 0,C 180,E1 -725.364,E2 -725.364} C_VEL
LIN {X 0,Y 601.442,Z 712.377,A -85,B 0,C 180,E1 -728.061,E2 -728.061} C_VEL
LIN {X 0,Y 601.431,Z 712.374,A -85,B 0,C 180,E1 -731.014,E2 -731.014} C_VEL
LIN {X 0,Y 601.418,Z 712.381,A -85,B 0,C 180,E1 -733.516,E2 -733.516} C_VEL
LIN {X 0,Y 601.443,Z 712.376,A -85,B 0,C 180,E1 -736.287,E2 -736.287} C_VEL
LIN {X 0,Y 601.42,Z 712.375,A -85,B 0,C 180,E1 -739.099,E2 -739.099} C_VEL
LIN {X 0,Y 601.408,Z 712.377,A -85,B 0,C 180,E1 -741.239,E2 -741.239} C_VEL
LIN {X 0,Y 601.461,Z 712.379,A -85,B 0,C 180,E1 -744.14,E2 -744.14} C_VEL
LIN {X 0,Y 601.454,Z 712.371,A -85,B 0,C 180,E1 -747.111,E2 -747.111} C_VEL
LIN {X 0,Y 601.421,Z 712.375,A -85,B 0,C 180,E1 -749.393,E2 -749.393} C_VEL
LIN {X 0,Y 601.414,Z 712.38,A -85,B 0,C 180,E1 -751.726,E2 -751.726} C_VEL
LIN {X 0,Y 601.433,Z 712.383,A -85,B 0,C 180,E1 -754.118,E2 -754.118} C_VEL
LIN {X 0,Y 601.413,Z 712.38,A -85,B 0,C 180,E1 -756.582,E2 -756.582} C_VEL
LIN {X 0,Y 601.442,Z 712.371,A -85,B 0,C 180,E1 -759.536,E2 -759.536} C_VEL
LIN {X 0,Y 601.419,Z 712.382,A -85,B 0,C 180,E1 -762.591,E2 -762.591} C_VEL
LIN {X 0,Y 601.427,Z 712.374,A -85,B 0,C 180,E1 -765.482,E2 -765.482} C_VEL
LIN {X 0,Y 601.428,Z 712.384,A -85,B 0,C 180,E1 -768.406,E2 -768.406} C_VEL
LIN {X 0,Y 601.435,Z 712.378,A -85,B 0,C 180,E1 -770.875,E2 -770.875} C_VEL
LIN {X 0,Y 601.444,Z 712.372,A -85,B 0,C 180,E1 -773.734,E2 -773.734} C_VEL
LIN {X 0,Y 601.437,Z 712.375,A -85,B 0,C 180,E1 -776.064,E2 -776.064} C_VEL
LIN {X 0,Y 601.443,Z 712.381,A -85,B 0,C 180,E1 -778.542,E2 -778.542} C_VEL
LIN {X 0,Y 601.433,Z 712.375,A -85,B 0,C 180,E1 -781.373,E2 -781.373} C_VEL
LIN {X 0,Y 601.421,Z 712.376,A -85,B 0,C 180,E1 -784.131,E2 -784.131} C_VEL
LIN {X 0,Y 601.42,Z 712.382,A -85,B 0,C 180,E1 -786.59,E2 -786.59} C_VEL
LIN {X 0,Y 601.449,Z 712.538,A -85,B 0,C 180,E1 -788.762,E2 -788.762} C_VEL
LIN {X 0,Y 601.521,Z 724.331,A -85,B 0,C 180,E1 -790.727,E2 -790.727} C_VEL
LIN {X 0,Y 601.494,Z 742.716,A -85,B 0,C 180,E1 -793.715,E2 -793.715} C_VEL
LIN {X 0,Y 601.44,Z 761.1,A -85,B 0,C 180,E1 -796.657,E2 -796.657} C_VEL
LIN {X 0,Y 601.388,Z 778.403,A -85,B 0,C 180,E1 -799.394,E2 -799.394} C_VEL
LIN {X 0,Y 601.429,Z 780.233,A -85,B 0,C 180,E1 -799.628,E2 -799.628} C_VEL
LIN {X 0,Y 601.535,Z 794.818,A -85,B 0,C 180,E1 -799.822,E2 -799.822} C_VEL
LIN {X 0,Y 601.504,Z 857.441,A -85,B 0,C 180,E1 -800.585,E2 -800.585} C_VEL
LIN {X 0,Y 601.514,Z 867.904,A -85,B 0,C 180,E1 -800.819,E2 -800.819} C_VEL
LIN {X 0,Y 601.472,Z 878.616,A -85,B 0,C 180,E1 -801.178,E2 -801.178} C_VEL
LIN {X 0,Y 601.446,Z 889.234,A -85,B 0,C 180,E1 -801.686,E2 -801.686} C_VEL
LIN {X 0,Y 601.413,Z 897.543,A -85,B 0,C 180,E1 -802.192,E2 -802.192} C_VEL
LIN {X 0,Y 601.414,Z 905.401,A -85,B 0,C 180,E1 -802.783,E2 -802.783} C_VEL
LIN {X 0,Y 601.412,Z 912.597,A -85,B 0,C 180,E1 -803.443,E2 -803.443} C_VEL
LIN {X 0,Y 601.391,Z 920.191,A -85,B 0,C 180,E1 -804.299,E2 -804.299} C_VEL
LIN {X 0,Y 601.38,Z 926.027,A -85,B 0,C 180,E1 -805.14,E2 -805.14} C_VEL
LIN {X 0,Y 601.344,Z 930.631,A -85,B 0,C 180,E1 -805.979,E2 -805.979} C_VEL
LIN {X 0,Y 601.344,Z 933.621,A -85,B 0,C 180,E1 -806.65,E2 -806.65} C_VEL
LIN {X 0,Y 601.326,Z 935.931,A -85,B 0,C 180,E1 -807.32,E2 -807.32} C_VEL
LIN {X 0,Y 601.339,Z 937.679,A -85,B 0,C 180,E1 -807.991,E2 -807.991} C_VEL
LIN {X 0,Y 601.346,Z 938.934,A -85,B 0,C 180,E1 -808.661,E2 -808.661} C_VEL
LIN {X 0,Y 601.337,Z 939.714,A -85,B 0,C 180,E1 -809.33,E2 -809.33} C_VEL
LIN {X 0,Y 601.332,Z 940,A -85,B 0,C 180,E1 -810,E2 -810} C_VEL
LIN {X 0,Y 601.337,Z 939.714,A -85,B 0,C 180,E1 -810.67,E2 -810.67} C_VEL
LIN {X 0,Y 601.346,Z 938.934,A -85,B 0,C 180,E1 -811.339,E2 -811.339} C_VEL
LIN {X 0,Y 601.339,Z 937.678,A -85,B 0,C 180,E1 -812.009,E2 -812.009} C_VEL
LIN {X 0,Y 601.343,Z 934.786,A -85,B 0,C 180,E1 -813.015,E2 -813.015} C_VEL
LIN {X 0,Y 601.364,Z 932.146,A -85,B 0,C 180,E1 -813.685,E2 -813.685} C_VEL
LIN {X 0,Y 601.341,Z 926.985,A -85,B 0,C 180,E1 -814.693,E2 -814.693} C_VEL
LIN {X 0,Y 601.383,Z 921.43,A -85,B 0,C 180,E1 -815.533,E2 -815.533} C_VEL
LIN {X 0,Y 601.393,Z 914.152,A -85,B 0,C 180,E1 -816.403,E2 -816.403} C_VEL
LIN {X 0,Y 601.416,Z 906.415,A -85,B 0,C 180,E1 -817.132,E2 -817.132} C_VEL
LIN {X 0,Y 601.433,Z 898.761,A -85,B 0,C 180,E1 -817.723,E2 -817.723} C_VEL
LIN {X 0,Y 601.454,Z 890.72,A -85,B 0,C 180,E1 -818.23,E2 -818.23} C_VEL
LIN {X 0,Y 601.481,Z 882.39,A -85,B 0,C 180,E1 -818.652,E2 -818.652} C_VEL
LIN {X 0,Y 601.473,Z 873.888,A -85,B 0,C 180,E1 -818.991,E2 -818.991} C_VEL
LIN {X 0,Y 601.511,Z 863.753,A -85,B 0,C 180,E1 -819.287,E2 -819.287} C_VEL
LIN {X 0,Y 601.515,Z 852.057,A -85,B 0,C 180,E1 -819.499,E2 -819.499} C_VEL
LIN {X 0,Y 601.503,Z 780.98,A -85,B 0,C 180,E1 -820.349,E2 -820.349} C_VEL
LIN {X 0,Y 601.414,Z 779.533,A -85,B 0,C 180,E1 -820.436,E2 -820.436} C_VEL
LIN {X 0,Y 601.44,Z 761.1,A -85,B 0,C 180,E1 -823.343,E2 -823.343} C_VEL
LIN {X 0,Y 601.494,Z 742.715,A -85,B 0,C 180,E1 -826.285,E2 -826.285} C_VEL
LIN {X 0,Y 601.521,Z 724.331,A -85,B 0,C 180,E1 -829.273,E2 -829.273} C_VEL
LIN {X 0,Y 601.45,Z 712.529,A -85,B 0,C 180,E1 -831.238,E2 -831.238} C_VEL
LIN {X 0,Y 601.455,Z 712.371,A -85,B 0,C 180,E1 -834.14,E2 -834.14} C_VEL
LIN {X 0,Y 601.446,Z 712.381,A -85,B 0,C 180,E1 -837.111,E2 -837.111} C_VEL
LIN {X 0,Y 601.427,Z 712.383,A -85,B 0,C 180,E1 -839.393,E2 -839.393} C_VEL
LIN {X 0,Y 601.415,Z 712.38,A -85,B 0,C 180,E1 -841.726,E2 -841.726} C_VEL
LIN {X 0,Y 601.433,Z 712.374,A -85,B 0,C 180,E1 -844.118,E2 -844.118} C_VEL
LIN {X 0,Y 601.411,Z 712.376,A -85,B 0,C 180,E1 -846.582,E2 -846.582} C_VEL
LIN {X 0,Y 601.441,Z 712.383,A -85,B 0,C 180,E1 -849.536,E2 -849.536} C_VEL
LIN {X 0,Y 601.43,Z 712.38,A -85,B 0,C 180,E1 -851.765,E2 -851.765} C_VEL
LIN {X 0,Y 601.426,Z 712.374,A -85,B 0,C 180,E1 -854.535,E2 -854.535} C_VEL
LIN {X 0,Y 601.419,Z 712.382,A -85,B 0,C 180,E1 -857.409,E2 -857.409} C_VEL
LIN {X 0,Y 601.443,Z 712.371,A -85,B 0,C 180,E1 -860.464,E2 -860.464} C_VEL
LIN {X 0,Y 601.413,Z 712.38,A -85,B 0,C 180,E1 -863.418,E2 -863.418} C_VEL
LIN {X 0,Y 601.437,Z 712.38,A -85,B 0,C 180,E1 -866.064,E2 -866.064} C_VEL
LIN {X 0,Y 601.434,Z 712.374,A -85,B 0,C 180,E1 -869.059,E2 -869.059} C_VEL
LIN {X 0,Y 601.43,Z 712.376,A -85,B 0,C 180,E1 -871.373,E2 -871.373} C_VEL
LIN {X 0,Y 601.401,Z 712.383,A -85,B 0,C 180,E1 -873.636,E2 -873.636} C_VEL
LIN {X 0,Y 601.422,Z 712.377,A -85,B 0,C 180,E1 -876.59,E2 -876.59} C_VEL
LIN {X 0,Y 601.435,Z 712.374,A -85,B 0,C 180,E1 -879.478,E2 -879.478} C_VEL
LIN {X 0,Y 601.4,Z 712.386,A -85,B 0,C 180,E1 -882.312,E2 -882.312} C_VEL
LIN {X 0,Y 601.414,Z 712.383,A -85,B 0,C 180,E1 -884.409,E2 -884.409} C_VEL
LIN {X 0,Y 601.421,Z 712.374,A -85,B 0,C 180,E1 -887.172,E2 -887.172} C_VEL
LIN {X 0,Y 601.433,Z 712.377,A -85,B 0,C 180,E1 -889.905,E2 -889.905} C_VEL
LIN {X 0,Y 601.44,Z 712.379,A -85,B 0,C 180,E1 -892.615,E2 -892.615} C_VEL
LIN {X 0,Y 601.431,Z 712.373,A -85,B 0,C 180,E1 -895.308,E2 -895.308} C_VEL
LIN {X 0,Y 601.429,Z 712.376,A -85,B 0,C 180,E1 -897.991,E2 -897.991} C_VEL
LIN {X 0,Y 601.451,Z 712.38,A -85,B 0,C 180,E1 -900.67,E2 -900.67} C_VEL
LIN {X 0,Y 601.426,Z 712.375,A -85,B 0,C 180,E1 -903.35,E2 -903.35} C_VEL
LIN {X 0,Y 601.44,Z 712.374,A -85,B 0,C 180,E1 -906.037,E2 -906.037} C_VEL
LIN {X 0,Y 601.417,Z 712.386,A -85,B 0,C 180,E1 -908.738,E2 -908.738} C_VEL
LIN {X 0,Y 601.415,Z 712.377,A -85,B 0,C 180,E1 -911.459,E2 -911.459} C_VEL
LIN {X 0,Y 601.411,Z 712.38,A -85,B 0,C 180,E1 -912.372,E2 -912.372} C_VEL
LIN {X 0,Y 600.742,Z 712.47,A -85,B 0,C 180,E1 -912.932,E2 -912.932} C_VEL
LIN {X 0,Y 597.89,Z 712.827,A -85,B 0,C 180,E1 -913.839,E2 -913.839} C_VEL
LIN {X 0,Y 595.48,Z 713.124,A -85,B 0,C 180,E1 -914.57,E2 -914.57} C_VEL
LIN {X 0,Y 594.443,Z 713.25,A -85,B 0,C 180,E1 -915.133,E2 -915.133} C_VEL
LIN {X 0,Y 594.358,Z 713.257,A -85,B 0,C 180,E1 -915.324,E2 -915.324} C_VEL
LIN {X 0,Y 594.389,Z 713.255,A -85,B 0,C 180,E1 -917.193,E2 -917.193} C_VEL
LIN {X 0,Y 594.376,Z 713.253,A -85,B 0,C 180,E1 -920.054,E2 -920.054} C_VEL
LIN {X 0,Y 594.358,Z 713.266,A -85,B 0,C 180,E1 -922.968,E2 -922.968} C_VEL
LIN {X 0,Y 594.365,Z 713.261,A -85,B 0,C 180,E1 -925.194,E2 -925.194} C_VEL
LIN {X 0,Y 594.388,Z 713.254,A -85,B 0,C 180,E1 -927.527,E2 -927.527} C_VEL
LIN {X 0,Y 594.372,Z 713.254,A -85,B 0,C 180,E1 -930.326,E2 -930.326} C_VEL
LIN {X 0,Y 594.38,Z 713.258,A -85,B 0,C 180,E1 -932.95,E2 -932.95} C_VEL
LIN {X 0,Y 594.351,Z 713.264,A -85,B 0,C 180,E1 -935.409,E2 -935.409} C_VEL
LIN {X 0,Y 594.377,Z 713.254,A -85,B 0,C 180,E1 -937.941,E2 -937.941} C_VEL
LIN {X 0,Y 594.376,Z 713.254,A -85,B 0,C 180,E1 -940.822,E2 -940.822} C_VEL
LIN {X 0,Y 594.368,Z 713.26,A -85,B 0,C 180,E1 -943.3,E2 -943.3} C_VEL
LIN {X 0,Y 594.361,Z 713.255,A -85,B 0,C 180,E1 -946.161,E2 -946.161} C_VEL
LIN {X 0,Y 594.375,Z 713.253,A -85,B 0,C 180,E1 -948.536,E2 -948.536} C_VEL
LIN {X 0,Y 594.382,Z 713.257,A -85,B 0,C 180,E1 -951.296,E2 -951.296} C_VEL
LIN {X 0,Y 594.35,Z 713.265,A -85,B 0,C 180,E1 -953.755,E2 -953.755} C_VEL
LIN {X 0,Y 594.356,Z 713.257,A -85,B 0,C 180,E1 -956.237,E2 -956.237} C_VEL
LIN {X 0,Y 594.366,Z 713.253,A -85,B 0,C 180,E1 -958.649,E2 -958.649} C_VEL
LIN {X 0,Y 594.384,Z 713.253,A -85,B 0,C 180,E1 -961.042,E2 -961.042} C_VEL
LIN {X 0,Y 594.357,Z 713.262,A -85,B 0,C 180,E1 -964.055,E2 -964.055} C_VEL
LIN {X 0,Y 594.37,Z 713.257,A -85,B 0,C 180,E1 -966.295,E2 -966.295} C_VEL
LIN {X 0,Y 594.404,Z 713.251,A -85,B 0,C 180,E1 -969.224,E2 -969.224} C_VEL
LIN {X 0,Y 594.394,Z 713.349,A -85,B 0,C 180,E1 -971.918,E2 -971.918} C_VEL
LIN {X 0,Y 594.345,Z 724.588,A -85,B 0,C 180,E1 -974.218,E2 -974.218} C_VEL
LIN {X 0,Y 594.326,Z 738.515,A -85,B 0,C 180,E1 -977.016,E2 -977.016} C_VEL
LIN {X 0,Y 594.299,Z 751.248,A -85,B 0,C 180,E1 -979.524,E2 -979.524} C_VEL
LIN {X 0,Y 594.518,Z 753.108,A -85,B 0,C 180,E1 -979.603,E2 -979.603} C_VEL
LIN {X 0,Y 594.519,Z 827.319,A -85,B 0,C 180,E1 -980.517,E2 -980.517} C_VEL
LIN {X 0,Y 594.489,Z 837.828,A -85,B 0,C 180,E1 -980.752,E2 -980.752} C_VEL
LIN {X 0,Y 594.458,Z 849.552,A -85,B 0,C 180,E1 -981.159,E2 -981.159} C_VEL
LIN {X 0,Y 594.431,Z 859.942,A -85,B 0,C 180,E1 -981.672,E2 -981.672} C_VEL
LIN {X 0,Y 594.372,Z 868.123,A -85,B 0,C 180,E1 -982.185,E2 -982.185} C_VEL
LIN {X 0,Y 594.356,Z 875.883,A -85,B 0,C 180,E1 -982.783,E2 -982.783} C_VEL
LIN {X 0,Y 594.345,Z 883.713,A -85,B 0,C 180,E1 -983.522,E2 -983.522} C_VEL
LIN {X 0,Y 594.308,Z 891.119,A -85,B 0,C 180,E1 -984.401,E2 -984.401} C_VEL
LIN {X 0,Y 594.255,Z 896.732,A -85,B 0,C 180,E1 -985.251,E2 -985.251} C_VEL
LIN {X 0,Y 594.286,Z 901.946,A -85,B 0,C 180,E1 -986.271,E2 -986.271} C_VEL
LIN {X 0,Y 594.248,Z 904.636,A -85,B 0,C 180,E1 -986.949,E2 -986.949} C_VEL
LIN {X 0,Y 594.241,Z 907.574,A -85,B 0,C 180,E1 -987.967,E2 -987.967} C_VEL
LIN {X 0,Y 594.244,Z 908.872,A -85,B 0,C 180,E1 -988.645,E2 -988.645} C_VEL
LIN {X 0,Y 594.235,Z 909.692,A -85,B 0,C 180,E1 -989.322,E2 -989.322} C_VEL
LIN {X 0,Y 594.234,Z 909.996,A -85,B 0,C 180,E1 -990,E2 -990} C_VEL
LIN {X 0,Y 594.236,Z 909.734,A -85,B 0,C 180,E1 -990.678,E2 -990.678} C_VEL
LIN {X 0,Y 594.246,Z 908.997,A -85,B 0,C 180,E1 -991.355,E2 -991.355} C_VEL
LIN {X 0,Y 594.242,Z 907.786,A -85,B 0,C 180,E1 -992.033,E2 -992.033} C_VEL
LIN {X 0,Y 594.247,Z 904.939,A -85,B 0,C 180,E1 -993.051,E2 -993.051} C_VEL
LIN {X 0,Y 594.286,Z 902.348,A -85,B 0,C 180,E1 -993.729,E2 -993.729} C_VEL
LIN {X 0,Y 594.265,Z 897.239,A -85,B 0,C 180,E1 -994.749,E2 -994.749} C_VEL
LIN {X 0,Y 594.309,Z 891.741,A -85,B 0,C 180,E1 -995.599,E2 -995.599} C_VEL
LIN {X 0,Y 594.343,Z 884.613,A -85,B 0,C 180,E1 -996.477,E2 -996.477} C_VEL
LIN {X 0,Y 594.354,Z 875.938,A -85,B 0,C 180,E1 -997.303,E2 -997.303} C_VEL
LIN {X 0,Y 594.378,Z 868.187,A -85,B 0,C 180,E1 -997.901,E2 -997.901} C_VEL
LIN {X 0,Y 594.42,Z 860.019,A -85,B 0,C 180,E1 -998.413,E2 -998.413} C_VEL
LIN {X 0,Y 594.46,Z 849.646,A -85,B 0,C 180,E1 -998.927,E2 -998.927} C_VEL
LIN {X 0,Y 594.489,Z 837.991,A -85,B 0,C 180,E1 -999.334,E2 -999.334} C_VEL
LIN {X 0,Y 594.552,Z 827.571,A -85,B 0,C 180,E1 -999.569,E2 -999.569} C_VEL
LIN {X 0,Y 594.51,Z 775.716,A -85,B 0,C 180,E1 -1000.214,E2 -1000.214} C_VEL
LIN {X 0,Y 594.397,Z 752.269,A -85,B 0,C 180,E1 -1000.506,E2 -1000.506} C_VEL
LIN {X 0,Y 594.303,Z 750.983,A -85,B 0,C 180,E1 -1000.605,E2 -1000.605} C_VEL
LIN {X 0,Y 594.357,Z 737.224,A -85,B 0,C 180,E1 -1003.331,E2 -1003.331} C_VEL
LIN {X 0,Y 594.391,Z 723.292,A -85,B 0,C 180,E1 -1006.133,E2 -1006.133} C_VEL
LIN {X 0,Y 594.401,Z 713.363,A -85,B 0,C 180,E1 -1008.171,E2 -1008.171} C_VEL
LIN {X 0,Y 594.374,Z 713.254,A -85,B 0,C 180,E1 -1010.915,E2 -1010.915} C_VEL
LIN {X 0,Y 594.364,Z 713.257,A -85,B 0,C 180,E1 -1013.705,E2 -1013.705} C_VEL
LIN {X 0,Y 594.357,Z 713.259,A -85,B 0,C 180,E1 -1016.701,E2 -1016.701} C_VEL
LIN {X 0,Y 594.381,Z 713.253,A -85,B 0,C 180,E1 -1018.999,E2 -1018.999} C_VEL
LIN {X 0,Y 594.372,Z 713.253,A -85,B 0,C 180,E1 -1021.641,E2 -1021.641} C_VEL
LIN {X 0,Y 594.379,Z 713.261,A -85,B 0,C 180,E1 -1024.58,E2 -1024.58} C_VEL
LIN {X 0,Y 594.386,Z 713.251,A -85,B 0,C 180,E1 -1027.608,E2 -1027.608} C_VEL
LIN {X 0,Y 594.363,Z 713.265,A -85,B 0,C 180,E1 -1030.568,E2 -1030.568} C_VEL
LIN {X 0,Y 594.367,Z 713.255,A -85,B 0,C 180,E1 -1033.3,E2 -1033.3} C_VEL
LIN {X 0,Y 594.361,Z 713.256,A -85,B 0,C 180,E1 -1036.161,E2 -1036.161} C_VEL
LIN {X 0,Y 594.377,Z 713.257,A -85,B 0,C 180,E1 -1038.536,E2 -1038.536} C_VEL
LIN {X 0,Y 594.372,Z 713.256,A -85,B 0,C 180,E1 -1041.297,E2 -1041.297} C_VEL
LIN {X 0,Y 594.35,Z 713.256,A -85,B 0,C 180,E1 -1043.755,E2 -1043.755} C_VEL
LIN {X 0,Y 594.366,Z 713.255,A -85,B 0,C 180,E1 -1046.238,E2 -1046.238} C_VEL
LIN {X 0,Y 594.369,Z 713.259,A -85,B 0,C 180,E1 -1048.65,E2 -1048.65} C_VEL
LIN {X 0,Y 594.385,Z 713.261,A -85,B 0,C 180,E1 -1051.042,E2 -1051.042} C_VEL
LIN {X 0,Y 594.376,Z 713.251,A -85,B 0,C 180,E1 -1053.979,E2 -1053.979} C_VEL
LIN {X 0,Y 594.376,Z 713.253,A -85,B 0,C 180,E1 -1056.295,E2 -1056.295} C_VEL
LIN {X 0,Y 594.409,Z 713.258,A -85,B 0,C 180,E1 -1059.225,E2 -1059.225} C_VEL
LIN {X 0,Y 594.353,Z 713.254,A -85,B 0,C 180,E1 -1062.095,E2 -1062.095} C_VEL
LIN {X 0,Y 594.365,Z 713.253,A -85,B 0,C 180,E1 -1064.219,E2 -1064.219} C_VEL
LIN {X 0,Y 594.38,Z 713.252,A -85,B 0,C 180,E1 -1066.321,E2 -1066.321} C_VEL
LIN {X 0,Y 594.377,Z 713.26,A -85,B 0,C 180,E1 -1069.095,E2 -1069.095} C_VEL
LIN {X 0,Y 594.419,Z 713.249,A -85,B 0,C 180,E1 -1071.843,E2 -1071.843} C_VEL
LIN {X 0,Y 594.391,Z 713.25,A -85,B 0,C 180,E1 -1074.572,E2 -1074.572} C_VEL
LIN {X 0,Y 594.412,Z 713.256,A -85,B 0,C 180,E1 -1077.289,E2 -1077.289} C_VEL
LIN {X 0,Y 594.415,Z 713.25,A -85,B 0,C 180,E1 -1080,E2 -1080} C_VEL
LIN {X 0,Y 594.414,Z 713.246,A -85,B 0,C 180,E1 -1082.711,E2 -1082.711} C_VEL
LIN {X 0,Y 594.387,Z 713.258,A -85,B 0,C 180,E1 -1085.428,E2 -1085.428} C_VEL
LIN {X 0,Y 594.419,Z 713.251,A -85,B 0,C 180,E1 -1088.157,E2 -1088.157} C_VEL
LIN {X 0,Y 594.395,Z 713.251,A -85,B 0,C 180,E1 -1091.075,E2 -1091.075} C_VEL
LIN {X 0,Y 594.384,Z 713.259,A -85,B 0,C 180,E1 -1093.679,E2 -1093.679} C_VEL
LIN {X 0,Y 594.399,Z 713.25,A -85,B 0,C 180,E1 -1096.72,E2 -1096.72} C_VEL
LIN {X 0,Y 594.37,Z 713.255,A -85,B 0,C 180,E1 -1099.334,E2 -1099.334} C_VEL
LIN {X 0,Y 594.368,Z 713.256,A -85,B 0,C 180,E1 -1101.503,E2 -1101.503} C_VEL
LIN {X 0,Y 594.391,Z 713.255,A -85,B 0,C 180,E1 -1104.446,E2 -1104.446} C_VEL
LIN {X 0,Y 594.386,Z 713.253,A -85,B 0,C 180,E1 -1106.699,E2 -1106.699} C_VEL
LIN {X 0,Y 594.383,Z 713.251,A -85,B 0,C 180,E1 -1108.998,E2 -1108.998} C_VEL
LIN {X 0,Y 594.393,Z 713.253,A -85,B 0,C 180,E1 -1111.645,E2 -1111.645} C_VEL
LIN {X 0,Y 594.4,Z 713.254,A -85,B 0,C 180,E1 -1114.579,E2 -1114.579} C_VEL
LIN {X 0,Y 594.387,Z 713.25,A -85,B 0,C 180,E1 -1117.086,E2 -1117.086} C_VEL
LIN {X 0,Y 594.377,Z 713.251,A -85,B 0,C 180,E1 -1119.774,E2 -1119.774} C_VEL
LIN {X 0,Y 594.374,Z 713.263,A -85,B 0,C 180,E1 -1122.375,E2 -1122.375} C_VEL
LIN {X 0,Y 594.365,Z 713.255,A -85,B 0,C 180,E1 -1125.191,E2 -1125.191} C_VEL
LIN {X 0,Y 594.388,Z 713.256,A -85,B 0,C 180,E1 -1128.151,E2 -1128.151} C_VEL
LIN {X 0,Y 594.388,Z 713.253,A -85,B 0,C 180,E1 -1131.195,E2 -1131.195} C_VEL
LIN {X 0,Y 594.397,Z 713.25,A -85,B 0,C 180,E1 -1133.759,E2 -1133.759} C_VEL
LIN {X 0,Y 594.383,Z 713.256,A -85,B 0,C 180,E1 -1136.239,E2 -1136.239} C_VEL
LIN {X 0,Y 594.392,Z 713.261,A -85,B 0,C 180,E1 -1138.651,E2 -1138.651} C_VEL
LIN {X 0,Y 594.385,Z 713.258,A -85,B 0,C 180,E1 -1141.042,E2 -1141.042} C_VEL
LIN {X 0,Y 594.393,Z 713.251,A -85,B 0,C 180,E1 -1143.976,E2 -1143.976} C_VEL
LIN {X 0,Y 594.39,Z 713.253,A -85,B 0,C 180,E1 -1146.296,E2 -1146.296} C_VEL
LIN {X 0,Y 594.452,Z 713.455,A -85,B 0,C 180,E1 -1148.657,E2 -1148.657} C_VEL
LIN {X 0,Y 594.57,Z 724.331,A -85,B 0,C 180,E1 -1150.493,E2 -1150.493} C_VEL
LIN {X 0,Y 594.488,Z 742.715,A -85,B 0,C 180,E1 -1153.517,E2 -1153.517} C_VEL
LIN {X 0,Y 594.412,Z 760.018,A -85,B 0,C 180,E1 -1156.322,E2 -1156.322} C_VEL
LIN {X 0,Y 594.32,Z 777.321,A -85,B 0,C 180,E1 -1159.094,E2 -1159.094} C_VEL
LIN {X 0,Y 594.378,Z 780.23,A -85,B 0,C 180,E1 -1159.504,E2 -1159.504} C_VEL
LIN {X 0,Y 594.563,Z 785.875,A -85,B 0,C 180,E1 -1159.593,E2 -1159.593} C_VEL
LIN {X 0,Y 594.544,Z 856.141,A -85,B 0,C 180,E1 -1160.453,E2 -1160.453} C_VEL
LIN {X 0,Y 594.511,Z 865.413,A -85,B 0,C 180,E1 -1160.645,E2 -1160.645} C_VEL
LIN {X 0,Y 594.464,Z 873.889,A -85,B 0,C 180,E1 -1160.902,E2 -1160.902} C_VEL
LIN {X 0,Y 594.446,Z 882.392,A -85,B 0,C 180,E1 -1161.244,E2 -1161.244} C_VEL
LIN {X 0,Y 594.431,Z 890.722,A -85,B 0,C 180,E1 -1161.672,E2 -1161.672} C_VEL
LIN {X 0,Y 594.369,Z 898.762,A -85,B 0,C 180,E1 -1162.185,E2 -1162.185} C_VEL
LIN {X 0,Y 594.357,Z 906.415,A -85,B 0,C 180,E1 -1162.783,E2 -1162.783} C_VEL
LIN {X 0,Y 594.33,Z 914.809,A -85,B 0,C 180,E1 -1163.589,E2 -1163.589} C_VEL
LIN {X 0,Y 594.309,Z 921.431,A -85,B 0,C 180,E1 -1164.401,E2 -1164.401} C_VEL
LIN {X 0,Y 594.256,Z 926.986,A -85,B 0,C 180,E1 -1165.251,E2 -1165.251} C_VEL
LIN {X 0,Y 594.286,Z 932.147,A -85,B 0,C 180,E1 -1166.271,E2 -1166.271} C_VEL
LIN {X 0,Y 594.246,Z 934.787,A -85,B 0,C 180,E1 -1166.949,E2 -1166.949} C_VEL
LIN {X 0,Y 594.239,Z 937.679,A -85,B 0,C 180,E1 -1167.967,E2 -1167.967} C_VEL
LIN {X 0,Y 594.246,Z 938.935,A -85,B 0,C 180,E1 -1168.645,E2 -1168.645} C_VEL
LIN {X 0,Y 594.237,Z 939.713,A -85,B 0,C 180,E1 -1169.322,E2 -1169.322} C_VEL
LIN {X 0,Y 594.233,Z 940,A -85,B 0,C 180,E1 -1170,E2 -1170} C_VEL
LIN {X 0,Y 594.237,Z 939.713,A -85,B 0,C 180,E1 -1170.678,E2 -1170.678} C_VEL
LIN {X 0,Y 594.246,Z 938.935,A -85,B 0,C 180,E1 -1171.355,E2 -1171.355} C_VEL
LIN {X 0,Y 594.239,Z 937.679,A -85,B 0,C 180,E1 -1172.033,E2 -1172.033} C_VEL
LIN {X 0,Y 594.246,Z 934.787,A -85,B 0,C 180,E1 -1173.051,E2 -1173.051} C_VEL
LIN {X 0,Y 594.286,Z 932.146,A -85,B 0,C 180,E1 -1173.729,E2 -1173.729} C_VEL
LIN {X 0,Y 594.256,Z 926.985,A -85,B 0,C 180,E1 -1174.749,E2 -1174.749} C_VEL
LIN {X 0,Y 594.309,Z 921.43,A -85,B 0,C 180,E1 -1175.599,E2 -1175.599} C_VEL
LIN {X 0,Y 594.344,Z 914.151,A -85,B 0,C 180,E1 -1176.479,E2 -1176.479} C_VEL
LIN {X 0,Y 594.357,Z 906.416,A -85,B 0,C 180,E1 -1177.217,E2 -1177.217} C_VEL
LIN {X 0,Y 594.369,Z 898.763,A -85,B 0,C 180,E1 -1177.815,E2 -1177.815} C_VEL
LIN {X 0,Y 594.431,Z 890.722,A -85,B 0,C 180,E1 -1178.328,E2 -1178.328} C_VEL
LIN {X 0,Y 594.446,Z 882.392,A -85,B 0,C 180,E1 -1178.756,E2 -1178.756} C_VEL
LIN {X 0,Y 594.464,Z 873.889,A -85,B 0,C 180,E1 -1179.098,E2 -1179.098} C_VEL
LIN {X 0,Y 594.518,Z 863.753,A -85,B 0,C 180,E1 -1179.397,E2 -1179.397} C_VEL
LIN {X 0,Y 594.535,Z 852.057,A -85,B 0,C 180,E1 -1179.612,E2 -1179.612} C_VEL
LIN {X 0,Y 594.459,Z 781.03,A -85,B 0,C 180,E1 -1180.473,E2 -1180.473} C_VEL
LIN {X 0,Y 594.355,Z 779.685,A -85,B 0,C 180,E1 -1180.539,E2 -1180.539} C_VEL
LIN {X 0,Y 594.418,Z 761.1,A -85,B 0,C 180,E1 -1183.504,E2 -1183.504} C_VEL
LIN {X 0,Y 594.486,Z 743.797,A -85,B 0,C 180,E1 -1186.306,E2 -1186.306} C_VEL
LIN {X 0,Y 594.54,Z 726.811,A -85,B 0,C 180,E1 -1189.097,E2 -1189.097} C_VEL
LIN {X 0,Y 594.487,Z 713.832,A -85,B 0,C 180,E1 -1191.264,E2 -1191.264} C_VEL
LIN {X 0,Y 594.436,Z 713.283,A -85,B 0,C 180,E1 -1191.422,E2 -1191.422} C_VEL
LIN {X 0,Y 594.39,Z 713.252,A -85,B 0,C 180,E1 -1194.446,E2 -1194.446} C_VEL
LIN {X 0,Y 594.384,Z 713.254,A -85,B 0,C 180,E1 -1196.7,E2 -1196.7} C_VEL
LIN {X 0,Y 594.383,Z 713.258,A -85,B 0,C 180,E1 -1198.998,E2 -1198.998} C_VEL
LIN {X 0,Y 594.393,Z 713.256,A -85,B 0,C 180,E1 -1201.645,E2 -1201.645} C_VEL
LIN {X 0,Y 594.399,Z 713.25,A -85,B 0,C 180,E1 -1204.579,E2 -1204.579} C_VEL
LIN {X 0,Y 594.385,Z 713.256,A -85,B 0,C 180,E1 -1207.087,E2 -1207.087} C_VEL
LIN {X 0,Y 594.378,Z 713.258,A -85,B 0,C 180,E1 -1209.775,E2 -1209.775} C_VEL
LIN {X 0,Y 594.371,Z 713.253,A -85,B 0,C 180,E1 -1212.375,E2 -1212.375} C_VEL
LIN {X 0,Y 594.365,Z 713.258,A -85,B 0,C 180,E1 -1215.191,E2 -1215.191} C_VEL
LIN {X 0,Y 594.386,Z 713.253,A -85,B 0,C 180,E1 -1218.151,E2 -1218.151} C_VEL
LIN {X 0,Y 594.39,Z 713.25,A -85,B 0,C 180,E1 -1221.196,E2 -1221.196} C_VEL
LIN {X 0,Y 594.397,Z 713.26,A -85,B 0,C 180,E1 -1223.759,E2 -1223.759} C_VEL
LIN {X 0,Y 594.383,Z 713.256,A -85,B 0,C 180,E1 -1226.239,E2 -1226.239} C_VEL
LIN {X 0,Y 594.392,Z 713.251,A -85,B 0,C 180,E1 -1228.651,E2 -1228.651} C_VEL
LIN {X 0,Y 594.385,Z 713.251,A -85,B 0,C 180,E1 -1231.042,E2 -1231.042} C_VEL
LIN {X 0,Y 594.384,Z 713.263,A -85,B 0,C 180,E1 -1233.978,E2 -1233.978} C_VEL
LIN {X 0,Y 594.392,Z 713.256,A -85,B 0,C 180,E1 -1236.296,E2 -1236.296} C_VEL
LIN {X 0,Y 594.409,Z 713.248,A -85,B 0,C 180,E1 -1239.225,E2 -1239.225} C_VEL
LIN {X 0,Y 594.382,Z 713.262,A -85,B 0,C 180,E1 -1242.096,E2 -1242.096} C_VEL
LIN {X 0,Y 594.37,Z 713.264,A -85,B 0,C 180,E1 -1244.219,E2 -1244.219} C_VEL
LIN {X 0,Y 594.383,Z 713.26,A -85,B 0,C 180,E1 -1246.321,E2 -1246.321} C_VEL
LIN {X 0,Y 594.381,Z 713.252,A -85,B 0,C 180,E1 -1249.095,E2 -1249.095} C_VEL
LIN {X 0,Y 594.418,Z 713.25,A -85,B 0,C 180,E1 -1251.843,E2 -1251.843} C_VEL
LIN {X 0,Y 594.388,Z 713.259,A -85,B 0,C 180,E1 -1254.572,E2 -1254.572} C_VEL
LIN {X 0,Y 594.414,Z 713.246,A -85,B 0,C 180,E1 -1257.289,E2 -1257.289} C_VEL
LIN {X 0,Y 594.416,Z 713.25,A -85,B 0,C 180,E1 -1260,E2 -1260} C_VEL
LIN {X 0,Y 594.414,Z 713.256,A -85,B 0,C 180,E1 -1262.711,E2 -1262.711} C_VEL
LIN {X 0,Y 594.392,Z 713.25,A -85,B 0,C 180,E1 -1265.428,E2 -1265.428} C_VEL
LIN {X 0,Y 594.419,Z 713.248,A -85,B 0,C 180,E1 -1268.157,E2 -1268.157} C_VEL
LIN {X 0,Y 594.393,Z 713.256,A -85,B 0,C 180,E1 -1271.074,E2 -1271.074} C_VEL
LIN {X 0,Y 594.381,Z 713.252,A -85,B 0,C 180,E1 -1273.679,E2 -1273.679} C_VEL
LIN {X 0,Y 594.358,Z 713.257,A -85,B 0,C 180,E1 -1275.324,E2 -1275.324} C_VEL
LIN {X 0,Y 593.685,Z 713.341,A -85,B 0,C 180,E1 -1275.89,E2 -1275.89} C_VEL
LIN {X 0,Y 590.82,Z 713.705,A -85,B 0,C 180,E1 -1276.808,E2 -1276.808} C_VEL
LIN {X 0,Y 588.41,Z 713.999,A -85,B 0,C 180,E1 -1277.547,E2 -1277.547} C_VEL
LIN {X 0,Y 587.387,Z 714.123,A -85,B 0,C 180,E1 -1278.117,E2 -1278.117} C_VEL
LIN {X 0,Y 587.31,Z 714.133,A -85,B 0,C 180,E1 -1278.31,E2 -1278.31} C_VEL
LIN {X 0,Y 587.333,Z 714.14,A -85,B 0,C 180,E1 -1281.038,E2 -1281.038} C_VEL
LIN {X 0,Y 587.315,Z 714.138,A -85,B 0,C 180,E1 -1283.259,E2 -1283.259} C_VEL
LIN {X 0,Y 587.326,Z 714.132,A -85,B 0,C 180,E1 -1285.517,E2 -1285.517} C_VEL
LIN {X 0,Y 587.35,Z 714.128,A -85,B 0,C 180,E1 -1287.818,E2 -1287.818} C_VEL
LIN {X 0,Y 587.328,Z 714.132,A -85,B 0,C 180,E1 -1290.508,E2 -1290.508} C_VEL
LIN {X 0,Y 587.34,Z 714.138,A -85,B 0,C 180,E1 -1293.112,E2 -1293.112} C_VEL
LIN {X 0,Y 587.291,Z 714.137,A -85,B 0,C 180,E1 -1295.9,E2 -1295.9} C_VEL
LIN {X 0,Y 587.32,Z 714.132,A -85,B 0,C 180,E1 -1298.48,E2 -1298.48} C_VEL
LIN {X 0,Y 587.336,Z 714.135,A -85,B 0,C 180,E1 -1301.157,E2 -1301.157} C_VEL
LIN {X 0,Y 587.313,Z 714.132,A -85,B 0,C 180,E1 -1304.112,E2 -1304.112} C_VEL
LIN {X 0,Y 587.316,Z 714.135,A -85,B 0,C 180,E1 -1306.994,E2 -1306.994} C_VEL
LIN {X 0,Y 587.311,Z 714.139,A -85,B 0,C 180,E1 -1309.745,E2 -1309.745} C_VEL
LIN {X 0,Y 587.343,Z 714.128,A -85,B 0,C 180,E1 -1312.392,E2 -1312.392} C_VEL
LIN {X 0,Y 587.34,Z 714.141,A -85,B 0,C 180,E1 -1315.654,E2 -1315.654} C_VEL
LIN {X 0,Y 587.339,Z 714.131,A -85,B 0,C 180,E1 -1318.231,E2 -1318.231} C_VEL
LIN {X 0,Y 587.349,Z 714.128,A -85,B 0,C 180,E1 -1320.867,E2 -1320.867} C_VEL
LIN {X 0,Y 587.332,Z 714.141,A -85,B 0,C 180,E1 -1323.825,E2 -1323.825} C_VEL
LIN {X 0,Y 587.327,Z 714.14,A -85,B 0,C 180,E1 -1325.993,E2 -1325.993} C_VEL
LIN {X 0,Y 587.316,Z 714.138,A -85,B 0,C 180,E1 -1328.225,E2 -1328.225} C_VEL
LIN {X 0,Y 587.347,Z 714.131,A -85,B 0,C 180,E1 -1331.151,E2 -1331.151} C_VEL
LIN {X 0,Y 587.363,Z 714.22,A -85,B 0,C 180,E1 -1331.874,E2 -1331.874} C_VEL
LIN {X 0,Y 587.316,Z 724.591,A -85,B 0,C 180,E1 -1334.025,E2 -1334.025} C_VEL
LIN {X 0,Y 587.318,Z 736.777,A -85,B 0,C 180,E1 -1336.506,E2 -1336.506} C_VEL
LIN {X 0,Y 587.235,Z 751.288,A -85,B 0,C 180,E1 -1339.399,E2 -1339.399} C_VEL
LIN {X 0,Y 587.446,Z 753.063,A -85,B 0,C 180,E1 -1339.475,E2 -1339.475} C_VEL
LIN {X 0,Y 587.541,Z 827.353,A -85,B 0,C 180,E1 -1340.403,E2 -1340.403} C_VEL
LIN {X 0,Y 587.493,Z 837.851,A -85,B 0,C 180,E1 -1340.641,E2 -1340.641} C_VEL
LIN {X 0,Y 587.454,Z 849.562,A -85,B 0,C 180,E1 -1341.053,E2 -1341.053} C_VEL
LIN {X 0,Y 587.395,Z 859.955,A -85,B 0,C 180,E1 -1341.572,E2 -1341.572} C_VEL
LIN {X 0,Y 587.333,Z 868.133,A -85,B 0,C 180,E1 -1342.091,E2 -1342.091} C_VEL
LIN {X 0,Y 587.291,Z 875.89,A -85,B 0,C 180,E1 -1342.695,E2 -1342.695} C_VEL
LIN {X 0,Y 587.286,Z 883.719,A -85,B 0,C 180,E1 -1343.443,E2 -1343.443} C_VEL
LIN {X 0,Y 587.238,Z 891.123,A -85,B 0,C 180,E1 -1344.334,E2 -1344.334} C_VEL
LIN {X 0,Y 587.173,Z 896.735,A -85,B 0,C 180,E1 -1345.194,E2 -1345.194} C_VEL
LIN {X 0,Y 587.21,Z 901.949,A -85,B 0,C 180,E1 -1346.226,E2 -1346.226} C_VEL
LIN {X 0,Y 587.157,Z 904.638,A -85,B 0,C 180,E1 -1346.912,E2 -1346.912} C_VEL
LIN {X 0,Y 587.141,Z 907.576,A -85,B 0,C 180,E1 -1347.942,E2 -1347.942} C_VEL
LIN {X 0,Y 587.144,Z 908.874,A -85,B 0,C 180,E1 -1348.628,E2 -1348.628} C_VEL
LIN {X 0,Y 587.136,Z 909.692,A -85,B 0,C 180,E1 -1349.314,E2 -1349.314} C_VEL
LIN {X 0,Y 587.135,Z 909.996,A -85,B 0,C 180,E1 -1350,E2 -1350} C_VEL
LIN {X 0,Y 587.137,Z 909.734,A -85,B 0,C 180,E1 -1350.686,E2 -1350.686} C_VEL
LIN {X 0,Y 587.146,Z 908.997,A -85,B 0,C 180,E1 -1351.372,E2 -1351.372} C_VEL
LIN {X 0,Y 587.141,Z 907.785,A -85,B 0,C 180,E1 -1352.058,E2 -1352.058} C_VEL
LIN {X 0,Y 587.156,Z 904.938,A -85,B 0,C 180,E1 -1353.088,E2 -1353.088} C_VEL
LIN {X 0,Y 587.21,Z 902.346,A -85,B 0,C 180,E1 -1353.774,E2 -1353.774} C_VEL
LIN {X 0,Y 587.169,Z 897.236,A -85,B 0,C 180,E1 -1354.806,E2 -1354.806} C_VEL
LIN {X 0,Y 587.239,Z 891.738,A -85,B 0,C 180,E1 -1355.666,E2 -1355.666} C_VEL
LIN {X 0,Y 587.269,Z 883.747,A -85,B 0,C 180,E1 -1356.644,E2 -1356.644} C_VEL
LIN {X 0,Y 587.295,Z 875.932,A -85,B 0,C 180,E1 -1357.391,E2 -1357.391} C_VEL
LIN {X 0,Y 587.341,Z 868.182,A -85,B 0,C 180,E1 -1357.996,E2 -1357.996} C_VEL
LIN {X 0,Y 587.395,Z 860.012,A -85,B 0,C 180,E1 -1358.515,E2 -1358.515} C_VEL
LIN {X 0,Y 587.458,Z 849.632,A -85,B 0,C 180,E1 -1359.034,E2 -1359.034} C_VEL
LIN {X 0,Y 587.499,Z 837.972,A -85,B 0,C 180,E1 -1359.446,E2 -1359.446} C_VEL
LIN {X 0,Y 587.562,Z 828.838,A -85,B 0,C 180,E1 -1359.662,E2 -1359.662} C_VEL
LIN {X 0,Y 587.535,Z 806.083,A -85,B 0,C 180,E1 -1359.967,E2 -1359.967} C_VEL
LIN {X 0,Y 587.418,Z 752.997,A -85,B 0,C 180,E1 -1360.619,E2 -1360.619} C_VEL
LIN {X 0,Y 587.249,Z 751.31,A -85,B 0,C 180,E1 -1360.687,E2 -1360.687} C_VEL
LIN {X 0,Y 587.323,Z 737.221,A -85,B 0,C 180,E1 -1363.494,E2 -1363.494} C_VEL
LIN {X 0,Y 587.367,Z 723.289,A -85,B 0,C 180,E1 -1366.331,E2 -1366.331} C_VEL
LIN {X 0,Y 587.377,Z 714.237,A -85,B 0,C 180,E1 -1368.215,E2 -1368.215} C_VEL
LIN {X 0,Y 587.333,Z 714.131,A -85,B 0,C 180,E1 -1371.038,E2 -1371.038} C_VEL
LIN {X 0,Y 587.308,Z 714.133,A -85,B 0,C 180,E1 -1373.259,E2 -1373.259} C_VEL
LIN {X 0,Y 587.315,Z 714.134,A -85,B 0,C 180,E1 -1375.518,E2 -1375.518} C_VEL
LIN {X 0,Y 587.323,Z 714.137,A -85,B 0,C 180,E1 -1378.597,E2 -1378.597} C_VEL
LIN {X 0,Y 587.323,Z 714.132,A -85,B 0,C 180,E1 -1380.967,E2 -1380.967} C_VEL
LIN {X 0,Y 587.324,Z 714.131,A -85,B 0,C 180,E1 -1383.397,E2 -1383.397} C_VEL
LIN {X 0,Y 587.29,Z 714.138,A -85,B 0,C 180,E1 -1385.9,E2 -1385.9} C_VEL
LIN {X 0,Y 587.326,Z 714.14,A -85,B 0,C 180,E1 -1388.48,E2 -1388.48} C_VEL
LIN {X 0,Y 587.334,Z 714.132,A -85,B 0,C 180,E1 -1391.157,E2 -1391.157} C_VEL
LIN {X 0,Y 587.313,Z 714.135,A -85,B 0,C 180,E1 -1394.112,E2 -1394.112} C_VEL
LIN {X 0,Y 587.314,Z 714.133,A -85,B 0,C 180,E1 -1396.993,E2 -1396.993} C_VEL
LIN {X 0,Y 587.309,Z 714.131,A -85,B 0,C 180,E1 -1399.745,E2 -1399.745} C_VEL
LIN {X 0,Y 587.342,Z 714.133,A -85,B 0,C 180,E1 -1402.392,E2 -1402.392} C_VEL
LIN {X 0,Y 587.345,Z 714.128,A -85,B 0,C 180,E1 -1405.653,E2 -1405.653} C_VEL
LIN {X 0,Y 587.342,Z 714.13,A -85,B 0,C 180,E1 -1408.231,E2 -1408.231} C_VEL
LIN {X 0,Y 587.35,Z 714.138,A -85,B 0,C 180,E1 -1410.867,E2 -1410.867} C_VEL
LIN {X 0,Y 587.338,Z 714.128,A -85,B 0,C 180,E1 -1413.824,E2 -1413.824} C_VEL
LIN {X 0,Y 587.33,Z 714.13,A -85,B 0,C 180,E1 -1415.993,E2 -1415.993} C_VEL
LIN {X 0,Y 587.322,Z 714.132,A -85,B 0,C 180,E1 -1418.226,E2 -1418.226} C_VEL
LIN {X 0,Y 587.351,Z 714.138,A -85,B 0,C 180,E1 -1421.151,E2 -1421.151} C_VEL
LIN {X 0,Y 587.325,Z 714.13,A -85,B 0,C 180,E1 -1424.025,E2 -1424.025} C_VEL
LIN {X 0,Y 587.359,Z 714.127,A -85,B 0,C 180,E1 -1426.154,E2 -1426.154} C_VEL
LIN {X 0,Y 587.343,Z 714.134,A -85,B 0,C 180,E1 -1428.962,E2 -1428.962} C_VEL
LIN {X 0,Y 587.37,Z 714.127,A -85,B 0,C 180,E1 -1431.745,E2 -1431.745} C_VEL
LIN {X 0,Y 587.359,Z 714.126,A -85,B 0,C 180,E1 -1434.507,E2 -1434.507} C_VEL
LIN {X 0,Y 587.377,Z 714.131,A -85,B 0,C 180,E1 -1437.257,E2 -1437.257} C_VEL
LIN {X 0,Y 587.384,Z 714.126,A -85,B 0,C 180,E1 -1440,E2 -1440} C_VEL
LIN {X 0,Y 587.379,Z 714.122,A -85,B 0,C 180,E1 -1442.743,E2 -1442.743} C_VEL
LIN {X 0,Y 587.353,Z 714.135,A -85,B 0,C 180,E1 -1445.493,E2 -1445.493} C_VEL
LIN {X 0,Y 587.372,Z 714.127,A -85,B 0,C 180,E1 -1448.255,E2 -1448.255} C_VEL
LIN {X 0,Y 587.351,Z 714.128,A -85,B 0,C 180,E1 -1451.134,E2 -1451.134} C_VEL
LIN {X 0,Y 587.368,Z 714.129,A -85,B 0,C 180,E1 -1454.26,E2 -1454.26} C_VEL
LIN {X 0,Y 587.36,Z 714.13,A -85,B 0,C 180,E1 -1457.406,E2 -1457.406} C_VEL
LIN {X 0,Y 587.333,Z 714.133,A -85,B 0,C 180,E1 -1460.305,E2 -1460.305} C_VEL
LIN {X 0,Y 587.325,Z 714.131,A -85,B 0,C 180,E1 -1463.259,E2 -1463.259} C_VEL
LIN {X 0,Y 587.335,Z 714.133,A -85,B 0,C 180,E1 -1465.517,E2 -1465.517} C_VEL
LIN {X 0,Y 587.351,Z 714.134,A -85,B 0,C 180,E1 -1467.818,E2 -1467.818} C_VEL
LIN {X 0,Y 587.344,Z 714.133,A -85,B 0,C 180,E1 -1470.511,E2 -1470.511} C_VEL
LIN {X 0,Y 587.338,Z 714.13,A -85,B 0,C 180,E1 -1473.396,E2 -1473.396} C_VEL
LIN {X 0,Y 587.358,Z 714.131,A -85,B 0,C 180,E1 -1475.895,E2 -1475.895} C_VEL
LIN {X 0,Y 587.335,Z 714.132,A -85,B 0,C 180,E1 -1478.479,E2 -1478.479} C_VEL
LIN {X 0,Y 587.339,Z 714.128,A -85,B 0,C 180,E1 -1481.157,E2 -1481.157} C_VEL
LIN {X 0,Y 587.328,Z 714.136,A -85,B 0,C 180,E1 -1484.113,E2 -1484.113} C_VEL
LIN {X 0,Y 587.316,Z 714.134,A -85,B 0,C 180,E1 -1486.994,E2 -1486.994} C_VEL
LIN {X 0,Y 587.322,Z 714.131,A -85,B 0,C 180,E1 -1489.746,E2 -1489.746} C_VEL
LIN {X 0,Y 587.346,Z 714.137,A -85,B 0,C 180,E1 -1492.392,E2 -1492.392} C_VEL
LIN {X 0,Y 587.353,Z 714.133,A -85,B 0,C 180,E1 -1494.946,E2 -1494.946} C_VEL
LIN {X 0,Y 587.341,Z 714.129,A -85,B 0,C 180,E1 -1497.421,E2 -1497.421} C_VEL
LIN {X 0,Y 587.337,Z 714.128,A -85,B 0,C 180,E1 -1499.83,E2 -1499.83} C_VEL
LIN {X 0,Y 587.352,Z 714.132,A -85,B 0,C 180,E1 -1502.307,E2 -1502.307} C_VEL
LIN {X 0,Y 587.34,Z 714.135,A -85,B 0,C 180,E1 -1504.484,E2 -1504.484} C_VEL
LIN {X 0,Y 587.342,Z 714.135,A -85,B 0,C 180,E1 -1507.486,E2 -1507.486} C_VEL
LIN {X 0,Y 587.395,Z 714.232,A -85,B 0,C 180,E1 -1508.505,E2 -1508.505} C_VEL
LIN {X 0,Y 587.624,Z 718.924,A -85,B 0,C 180,E1 -1509.34,E2 -1509.34} C_VEL
LIN {X 0,Y 587.498,Z 736.227,A -85,B 0,C 180,E1 -1512.239,E2 -1512.239} C_VEL
LIN {X 0,Y 587.414,Z 752.448,A -85,B 0,C 180,E1 -1514.917,E2 -1514.917} C_VEL
LIN {X 0,Y 587.335,Z 769.751,A -85,B 0,C 180,E1 -1517.737,E2 -1517.737} C_VEL
LIN {X 0,Y 587.298,Z 779.947,A -85,B 0,C 180,E1 -1519.355,E2 -1519.355} C_VEL
LIN {X 0,Y 587.582,Z 782.376,A -85,B 0,C 180,E1 -1519.426,E2 -1519.426} C_VEL
LIN {X 0,Y 587.564,Z 856.14,A -85,B 0,C 180,E1 -1520.338,E2 -1520.338} C_VEL
LIN {X 0,Y 587.502,Z 865.413,A -85,B 0,C 180,E1 -1520.533,E2 -1520.533} C_VEL
LIN {X 0,Y 587.447,Z 873.89,A -85,B 0,C 180,E1 -1520.792,E2 -1520.792} C_VEL
LIN {X 0,Y 587.418,Z 882.394,A -85,B 0,C 180,E1 -1521.139,E2 -1521.139} C_VEL
LIN {X 0,Y 587.395,Z 890.724,A -85,B 0,C 180,E1 -1521.572,E2 -1521.572} C_VEL
LIN {X 0,Y 587.336,Z 898.763,A -85,B 0,C 180,E1 -1522.091,E2 -1522.091} C_VEL
LIN {X 0,Y 587.291,Z 906.415,A -85,B 0,C 180,E1 -1522.695,E2 -1522.695} C_VEL
LIN {X 0,Y 587.281,Z 914.809,A -85,B 0,C 180,E1 -1523.512,E2 -1523.512} C_VEL
LIN {X 0,Y 587.238,Z 921.431,A -85,B 0,C 180,E1 -1524.334,E2 -1524.334} C_VEL
LIN {X 0,Y 587.17,Z 926.986,A -85,B 0,C 180,E1 -1525.194,E2 -1525.194} C_VEL
LIN {X 0,Y 587.21,Z 932.147,A -85,B 0,C 180,E1 -1526.226,E2 -1526.226} C_VEL
LIN {X 0,Y 587.155,Z 934.787,A -85,B 0,C 180,E1 -1526.912,E2 -1526.912} C_VEL
LIN {X 0,Y 587.138,Z 937.68,A -85,B 0,C 180,E1 -1527.942,E2 -1527.942} C_VEL
LIN {X 0,Y 587.146,Z 938.935,A -85,B 0,C 180,E1 -1528.628,E2 -1528.628} C_VEL
LIN {X 0,Y 587.137,Z 939.712,A -85,B 0,C 180,E1 -1529.314,E2 -1529.314} C_VEL
LIN {X 0,Y 587.134,Z 940,A -85,B 0,C 180,E1 -1530,E2 -1530} C_VEL
LIN {X 0,Y 587.137,Z 939.712,A -85,B 0,C 180,E1 -1530.686,E2 -1530.686} C_VEL
LIN {X 0,Y 587.146,Z 938.935,A -85,B 0,C 180,E1 -1531.372,E2 -1531.372} C_VEL
LIN {X 0,Y 587.138,Z 937.679,A -85,B 0,C 180,E1 -1532.058,E2 -1532.058} C_VEL
LIN {X 0,Y 587.155,Z 934.787,A -85,B 0,C 180,E1 -1533.088,E2 -1533.088} C_VEL
LIN {X 0,Y 587.21,Z 932.147,A -85,B 0,C 180,E1 -1533.774,E2 -1533.774} C_VEL
LIN {X 0,Y 587.17,Z 926.985,A -85,B 0,C 180,E1 -1534.806,E2 -1534.806} C_VEL
LIN {X 0,Y 587.238,Z 921.43,A -85,B 0,C 180,E1 -1535.666,E2 -1535.666} C_VEL
LIN {X 0,Y 587.269,Z 913.286,A -85,B 0,C 180,E1 -1536.645,E2 -1536.645} C_VEL
LIN {X 0,Y 587.291,Z 906.417,A -85,B 0,C 180,E1 -1537.305,E2 -1537.305} C_VEL
LIN {X 0,Y 587.336,Z 898.765,A -85,B 0,C 180,E1 -1537.909,E2 -1537.909} C_VEL
LIN {X 0,Y 587.395,Z 890.724,A -85,B 0,C 180,E1 -1538.428,E2 -1538.428} C_VEL
LIN {X 0,Y 587.418,Z 882.395,A -85,B 0,C 180,E1 -1538.861,E2 -1538.861} C_VEL
LIN {X 0,Y 587.447,Z 873.891,A -85,B 0,C 180,E1 -1539.208,E2 -1539.208} C_VEL
LIN {X 0,Y 587.512,Z 863.753,A -85,B 0,C 180,E1 -1539.511,E2 -1539.511} C_VEL
LIN {X 0,Y 587.558,Z 852.057,A -85,B 0,C 180,E1 -1539.727,E2 -1539.727} C_VEL
LIN {X 0,Y 587.426,Z 781.062,A -85,B 0,C 180,E1 -1540.599,E2 -1540.599} C_VEL
LIN {X 0,Y 587.302,Z 779.704,A -85,B 0,C 180,E1 -1540.666,E2 -1540.666} C_VEL
LIN {X 0,Y 587.379,Z 762.181,A -85,B 0,C 180,E1 -1543.492,E2 -1543.492} C_VEL
LIN {X 0,Y 587.491,Z 743.797,A -85,B 0,C 180,E1 -1546.506,E2 -1546.506} C_VEL
LIN {X 0,Y 587.579,Z 725.413,A -85,B 0,C 180,E1 -1549.567,E2 -1549.567} C_VEL
LIN {X 0,Y 587.615,Z 716.275,A -85,B 0,C 180,E1 -1551.109,E2 -1551.109} C_VEL
LIN {X 0,Y 587.367,Z 714.209,A -85,B 0,C 180,E1 -1551.496,E2 -1551.496} C_VEL
LIN {X 0,Y 587.354,Z 714.129,A -85,B 0,C 180,E1 -1554.58,E2 -1554.58} C_VEL
LIN {X 0,Y 587.33,Z 714.138,A -85,B 0,C 180,E1 -1557.046,E2 -1557.046} C_VEL
LIN {X 0,Y 587.35,Z 714.136,A -85,B 0,C 180,E1 -1559.379,E2 -1559.379} C_VEL
LIN {X 0,Y 587.356,Z 714.13,A -85,B 0,C 180,E1 -1561.837,E2 -1561.837} C_VEL
LIN {X 0,Y 587.358,Z 714.127,A -85,B 0,C 180,E1 -1564.349,E2 -1564.349} C_VEL
LIN {X 0,Y 587.354,Z 714.128,A -85,B 0,C 180,E1 -1566.747,E2 -1566.747} C_VEL
LIN {X 0,Y 587.347,Z 714.137,A -85,B 0,C 180,E1 -1569.359,E2 -1569.359} C_VEL
LIN {X 0,Y 587.336,Z 714.131,A -85,B 0,C 180,E1 -1572.108,E2 -1572.108} C_VEL
LIN {X 0,Y 587.317,Z 714.135,A -85,B 0,C 180,E1 -1575.089,E2 -1575.089} C_VEL
LIN {X 0,Y 587.354,Z 714.132,A -85,B 0,C 180,E1 -1577.928,E2 -1577.928} C_VEL
LIN {X 0,Y 587.336,Z 714.126,A -85,B 0,C 180,E1 -1581.058,E2 -1581.058} C_VEL
LIN {X 0,Y 587.355,Z 714.128,A -85,B 0,C 180,E1 -1583.292,E2 -1583.292} C_VEL
LIN {X 0,Y 587.37,Z 714.136,A -85,B 0,C 180,E1 -1585.781,E2 -1585.781} C_VEL
LIN {X 0,Y 587.353,Z 714.132,A -85,B 0,C 180,E1 -1588.232,E2 -1588.232} C_VEL
LIN {X 0,Y 587.351,Z 714.126,A -85,B 0,C 180,E1 -1590.867,E2 -1590.867} C_VEL
LIN {X 0,Y 587.36,Z 714.135,A -85,B 0,C 180,E1 -1593.819,E2 -1593.819} C_VEL
LIN {X 0,Y 587.34,Z 714.14,A -85,B 0,C 180,E1 -1595.994,E2 -1595.994} C_VEL
LIN {X 0,Y 587.324,Z 714.138,A -85,B 0,C 180,E1 -1598.226,E2 -1598.226} C_VEL
LIN {X 0,Y 587.353,Z 714.127,A -85,B 0,C 180,E1 -1601.151,E2 -1601.151} C_VEL
LIN {X 0,Y 587.356,Z 714.127,A -85,B 0,C 180,E1 -1603.311,E2 -1603.311} C_VEL
LIN {X 0,Y 587.361,Z 714.136,A -85,B 0,C 180,E1 -1606.154,E2 -1606.154} C_VEL
LIN {X 0,Y 587.346,Z 714.129,A -85,B 0,C 180,E1 -1608.963,E2 -1608.963} C_VEL
LIN {X 0,Y 587.372,Z 714.127,A -85,B 0,C 180,E1 -1611.745,E2 -1611.745} C_VEL
LIN {X 0,Y 587.354,Z 714.136,A -85,B 0,C 180,E1 -1614.507,E2 -1614.507} C_VEL
LIN {X 0,Y 587.38,Z 714.122,A -85,B 0,C 180,E1 -1617.257,E2 -1617.257} C_VEL
LIN {X 0,Y 587.386,Z 714.125,A -85,B 0,C 180,E1 -1620,E2 -1620} C_VEL
LIN {X 0,Y 587.38,Z 714.132,A -85,B 0,C 180,E1 -1622.743,E2 -1622.743} C_VEL
LIN {X 0,Y 587.36,Z 714.126,A -85,B 0,C 180,E1 -1625.493,E2 -1625.493} C_VEL
LIN {X 0,Y 587.37,Z 714.127,A -85,B 0,C 180,E1 -1628.255,E2 -1628.255} C_VEL
LIN {X 0,Y 587.351,Z 714.132,A -85,B 0,C 180,E1 -1631.134,E2 -1631.134} C_VEL
LIN {X 0,Y 587.368,Z 714.128,A -85,B 0,C 180,E1 -1634.26,E2 -1634.26} C_VEL
LIN {X 0,Y 587.35,Z 714.129,A -85,B 0,C 180,E1 -1637.406,E2 -1637.406} C_VEL
LIN {X 0,Y 587.31,Z 714.133,A -85,B 0,C 180,E1 -1638.31,E2 -1638.31} C_VEL
LIN {X 0,Y 586.667,Z 714.222,A -85,B 0,C 180,E1 -1638.882,E2 -1638.882} C_VEL
LIN {X 0,Y 583.844,Z 714.577,A -85,B 0,C 180,E1 -1639.81,E2 -1639.81} C_VEL
LIN {X 0,Y 581.434,Z 714.877,A -85,B 0,C 180,E1 -1640.557,E2 -1640.557} C_VEL
LIN {X 0,Y 580.381,Z 715.004,A -85,B 0,C 180,E1 -1641.134,E2 -1641.134} C_VEL
LIN {X 0,Y 580.285,Z 715.013,A -85,B 0,C 180,E1 -1641.329,E2 -1641.329} C_VEL
LIN {X 0,Y 580.299,Z 715.007,A -85,B 0,C 180,E1 -1644.316,E2 -1644.316} C_VEL
LIN {X 0,Y 580.29,Z 715.012,A -85,B 0,C 180,E1 -1647.402,E2 -1647.402} C_VEL
LIN {X 0,Y 580.28,Z 715.01,A -85,B 0,C 180,E1 -1649.773,E2 -1649.773} C_VEL
LIN {X 0,Y 580.301,Z 715.005,A -85,B 0,C 180,E1 -1652.2,E2 -1652.2} C_VEL
LIN {X 0,Y 580.29,Z 715.009,A -85,B 0,C 180,E1 -1654.696,E2 -1654.696} C_VEL
LIN {X 0,Y 580.298,Z 715.018,A -85,B 0,C 180,E1 -1657.269,E2 -1657.269} C_VEL
LIN {X 0,Y 580.289,Z 715.006,A -85,B 0,C 180,E1 -1660.27,E2 -1660.27} C_VEL
LIN {X 0,Y 580.279,Z 715.004,A -85,B 0,C 180,E1 -1662.706,E2 -1662.706} C_VEL
LIN {X 0,Y 580.256,Z 715.02,A -85,B 0,C 180,E1 -1665.611,E2 -1665.611} C_VEL
LIN {X 0,Y 580.278,Z 715.01,A -85,B 0,C 180,E1 -1668.231,E2 -1668.231} C_VEL
LIN {X 0,Y 580.278,Z 715.009,A -85,B 0,C 180,E1 -1670.965,E2 -1670.965} C_VEL
LIN {X 0,Y 580.27,Z 715.02,A -85,B 0,C 180,E1 -1673.596,E2 -1673.596} C_VEL
LIN {X 0,Y 580.28,Z 715.012,A -85,B 0,C 180,E1 -1676.143,E2 -1676.143} C_VEL
LIN {X 0,Y 580.273,Z 715.008,A -85,B 0,C 180,E1 -1678.614,E2 -1678.614} C_VEL
LIN {X 0,Y 580.292,Z 715.008,A -85,B 0,C 180,E1 -1681.024,E2 -1681.024} C_VEL
LIN {X 0,Y 580.27,Z 715.016,A -85,B 0,C 180,E1 -1684.15,E2 -1684.15} C_VEL
LIN {X 0,Y 580.27,Z 715.012,A -85,B 0,C 180,E1 -1686.442,E2 -1686.442} C_VEL
LIN {X 0,Y 580.273,Z 715.013,A -85,B 0,C 180,E1 -1689.437,E2 -1689.437} C_VEL
LIN {X 0,Y 580.311,Z 715.1,A -85,B 0,C 180,E1 -1691.829,E2 -1691.829} C_VEL
LIN {X 0,Y 580.298,Z 724.594,A -85,B 0,C 180,E1 -1693.826,E2 -1693.826} C_VEL
LIN {X 0,Y 580.243,Z 736.779,A -85,B 0,C 180,E1 -1696.338,E2 -1696.338} C_VEL
LIN {X 0,Y 580.186,Z 751.251,A -85,B 0,C 180,E1 -1699.261,E2 -1699.261} C_VEL
LIN {X 0,Y 580.344,Z 752.936,A -85,B 0,C 180,E1 -1699.341,E2 -1699.341} C_VEL
LIN {X 0,Y 580.619,Z 763.632,A -85,B 0,C 180,E1 -1699.481,E2 -1699.481} C_VEL
LIN {X 0,Y 580.548,Z 827.386,A -85,B 0,C 180,E1 -1700.286,E2 -1700.286} C_VEL
LIN {X 0,Y 580.499,Z 837.874,A -85,B 0,C 180,E1 -1700.527,E2 -1700.527} C_VEL
LIN {X 0,Y 580.436,Z 849.572,A -85,B 0,C 180,E1 -1700.944,E2 -1700.944} C_VEL
LIN {X 0,Y 580.362,Z 859.967,A -85,B 0,C 180,E1 -1701.469,E2 -1701.469} C_VEL
LIN {X 0,Y 580.285,Z 868.143,A -85,B 0,C 180,E1 -1701.994,E2 -1701.994} C_VEL
LIN {X 0,Y 580.24,Z 875.898,A -85,B 0,C 180,E1 -1702.606,E2 -1702.606} C_VEL
LIN {X 0,Y 580.21,Z 883.518,A -85,B 0,C 180,E1 -1703.342,E2 -1703.342} C_VEL
LIN {X 0,Y 580.173,Z 891.127,A -85,B 0,C 180,E1 -1704.264,E2 -1704.264} C_VEL
LIN {X 0,Y 580.088,Z 896.739,A -85,B 0,C 180,E1 -1705.135,E2 -1705.135} C_VEL
LIN {X 0,Y 580.137,Z 901.952,A -85,B 0,C 180,E1 -1706.18,E2 -1706.18} C_VEL
LIN {X 0,Y 580.072,Z 904.641,A -85,B 0,C 180,E1 -1706.875,E2 -1706.875} C_VEL
LIN {X 0,Y 580.04,Z 907.578,A -85,B 0,C 180,E1 -1707.917,E2 -1707.917} C_VEL
LIN {X 0,Y 580.044,Z 908.875,A -85,B 0,C 180,E1 -1708.611,E2 -1708.611} C_VEL
LIN {X 0,Y 580.036,Z 909.691,A -85,B 0,C 180,E1 -1709.306,E2 -1709.306} C_VEL
LIN {X 0,Y 580.036,Z 909.996,A -85,B 0,C 180,E1 -1710,E2 -1710} C_VEL
LIN {X 0,Y 580.037,Z 909.733,A -85,B 0,C 180,E1 -1710.694,E2 -1710.694} C_VEL
LIN {X 0,Y 580.046,Z 908.997,A -85,B 0,C 180,E1 -1711.389,E2 -1711.389} C_VEL
LIN {X 0,Y 580.041,Z 907.785,A -85,B 0,C 180,E1 -1712.083,E2 -1712.083} C_VEL
LIN {X 0,Y 580.071,Z 904.937,A -85,B 0,C 180,E1 -1713.125,E2 -1713.125} C_VEL
LIN {X 0,Y 580.122,Z 902.344,A -85,B 0,C 180,E1 -1713.82,E2 -1713.82} C_VEL
LIN {X 0,Y 580.075,Z 897.234,A -85,B 0,C 180,E1 -1714.865,E2 -1714.865} C_VEL
LIN {X 0,Y 580.173,Z 891.735,A -85,B 0,C 180,E1 -1715.736,E2 -1715.736} C_VEL
LIN {X 0,Y 580.195,Z 884.504,A -85,B 0,C 180,E1 -1716.646,E2 -1716.646} C_VEL
LIN {X 0,Y 580.253,Z 875.927,A -85,B 0,C 180,E1 -1717.481,E2 -1717.481} C_VEL
LIN {X 0,Y 580.308,Z 868.176,A -85,B 0,C 180,E1 -1718.093,E2 -1718.093} C_VEL
LIN {X 0,Y 580.377,Z 860.005,A -85,B 0,C 180,E1 -1718.618,E2 -1718.618} C_VEL
LIN {X 0,Y 580.437,Z 849.618,A -85,B 0,C 180,E1 -1719.144,E2 -1719.144} C_VEL
LIN {X 0,Y 580.498,Z 837.953,A -85,B 0,C 180,E1 -1719.561,E2 -1719.561} C_VEL
LIN {X 0,Y 580.571,Z 827.506,A -85,B 0,C 180,E1 -1719.801,E2 -1719.801} C_VEL
LIN {X 0,Y 580.625,Z 763.186,A -85,B 0,C 180,E1 -1720.614,E2 -1720.614} C_VEL
LIN {X 0,Y 580.459,Z 753.855,A -85,B 0,C 180,E1 -1720.732,E2 -1720.732} C_VEL
LIN {X 0,Y 580.212,Z 751.487,A -85,B 0,C 180,E1 -1720.803,E2 -1720.803} C_VEL
LIN {X 0,Y 580.212,Z 744.184,A -85,B 0,C 180,E1 -1722.238,E2 -1722.238} C_VEL
LIN {X 0,Y 580.29,Z 730.252,A -85,B 0,C 180,E1 -1725.093,E2 -1725.093} C_VEL
LIN {X 0,Y 580.385,Z 716.319,A -85,B 0,C 180,E1 -1727.986,E2 -1727.986} C_VEL
LIN {X 0,Y 580.351,Z 715.111,A -85,B 0,C 180,E1 -1728.261,E2 -1728.261} C_VEL
LIN {X 0,Y 580.285,Z 715.009,A -85,B 0,C 180,E1 -1731.305,E2 -1731.305} C_VEL
LIN {X 0,Y 580.291,Z 715.017,A -85,B 0,C 180,E1 -1734.317,E2 -1734.317} C_VEL
LIN {X 0,Y 580.248,Z 715.013,A -85,B 0,C 180,E1 -1737.404,E2 -1737.404} C_VEL
LIN {X 0,Y 580.277,Z 715.011,A -85,B 0,C 180,E1 -1739.773,E2 -1739.773} C_VEL
LIN {X 0,Y 580.298,Z 715.013,A -85,B 0,C 180,E1 -1742.201,E2 -1742.201} C_VEL
LIN {X 0,Y 580.287,Z 715.015,A -85,B 0,C 180,E1 -1744.696,E2 -1744.696} C_VEL
LIN {X 0,Y 580.297,Z 715.006,A -85,B 0,C 180,E1 -1747.269,E2 -1747.269} C_VEL
LIN {X 0,Y 580.288,Z 715.012,A -85,B 0,C 180,E1 -1750.27,E2 -1750.27} C_VEL
LIN {X 0,Y 580.279,Z 715.018,A -85,B 0,C 180,E1 -1752.706,E2 -1752.706} C_VEL
LIN {X 0,Y 580.256,Z 715.01,A -85,B 0,C 180,E1 -1755.611,E2 -1755.611} C_VEL
LIN {X 0,Y 580.277,Z 715.007,A -85,B 0,C 180,E1 -1758.231,E2 -1758.231} C_VEL
LIN {X 0,Y 580.272,Z 715.017,A -85,B 0,C 180,E1 -1760.964,E2 -1760.964} C_VEL
LIN {X 0,Y 580.269,Z 715.011,A -85,B 0,C 180,E1 -1763.596,E2 -1763.596} C_VEL
LIN {X 0,Y 580.302,Z 715.006,A -85,B 0,C 180,E1 -1766.144,E2 -1766.144} C_VEL
LIN {X 0,Y 580.275,Z 715.014,A -85,B 0,C 180,E1 -1768.614,E2 -1768.614} C_VEL
LIN {X 0,Y 580.293,Z 715.017,A -85,B 0,C 180,E1 -1771.024,E2 -1771.024} C_VEL
LIN {X 0,Y 580.291,Z 715.007,A -85,B 0,C 180,E1 -1773.667,E2 -1773.667} C_VEL
LIN {X 0,Y 580.299,Z 715.007,A -85,B 0,C 180,E1 -1775.684,E2 -1775.684} C_VEL
LIN {X 0,Y 580.287,Z 715.012,A -85,B 0,C 180,E1 -1778.695,E2 -1778.695} C_VEL
LIN {X 0,Y 580.3,Z 715.013,A -85,B 0,C 180,E1 -1780.913,E2 -1780.913} C_VEL
LIN {X 0,Y 580.281,Z 715.009,A -85,B 0,C 180,E1 -1783.826,E2 -1783.826} C_VEL
LIN {X 0,Y 580.327,Z 715.003,A -85,B 0,C 180,E1 -1785.983,E2 -1785.983} C_VEL
LIN {X 0,Y 580.308,Z 715.008,A -85,B 0,C 180,E1 -1788.827,E2 -1788.827} C_VEL
LIN {X 0,Y 580.332,Z 715.005,A -85,B 0,C 180,E1 -1791.644,E2 -1791.644} C_VEL
LIN {X 0,Y 580.327,Z 715.002,A -85,B 0,C 180,E1 -1794.44,E2 -1794.44} C_VEL
LIN {X 0,Y 580.343,Z 715.007,A -85,B 0,C 180,E1 -1797.223,E2 -1797.223} C_VEL
LIN {X 0,Y 580.353,Z 715.001,A -85,B 0,C 180,E1 -1800,E2 -1800} C_VEL
LIN {X 0,Y 580.345,Z 714.998,A -85,B 0,C 180,E1 -1802.776,E2 -1802.776} C_VEL
LIN {X 0,Y 580.32,Z 715.013,A -85,B 0,C 180,E1 -1805.56,E2 -1805.56} C_VEL
LIN {X 0,Y 580.336,Z 715.003,A -85,B 0,C 180,E1 -1808.356,E2 -1808.356} C_VEL
LIN {X 0,Y 580.303,Z 715.007,A -85,B 0,C 180,E1 -1811.191,E2 -1811.191} C_VEL
LIN {X 0,Y 580.328,Z 715.009,A -85,B 0,C 180,E1 -1814.017,E2 -1814.017} C_VEL
LIN {X 0,Y 580.315,Z 715.004,A -85,B 0,C 180,E1 -1816.914,E2 -1816.914} C_VEL
LIN {X 0,Y 580.308,Z 715.014,A -85,B 0,C 180,E1 -1819.822,E2 -1819.822} C_VEL
LIN {X 0,Y 580.297,Z 715.006,A -85,B 0,C 180,E1 -1822.802,E2 -1822.802} C_VEL
LIN {X 0,Y 580.308,Z 715.005,A -85,B 0,C 180,E1 -1825.08,E2 -1825.08} C_VEL
LIN {X 0,Y 580.303,Z 715.013,A -85,B 0,C 180,E1 -1828.185,E2 -1828.185} C_VEL
LIN {X 0,Y 580.295,Z 715.009,A -85,B 0,C 180,E1 -1830.696,E2 -1830.696} C_VEL
LIN {X 0,Y 580.306,Z 715.006,A -85,B 0,C 180,E1 -1833.316,E2 -1833.316} C_VEL
LIN {X 0,Y 580.328,Z 715.005,A -85,B 0,C 180,E1 -1835.767,E2 -1835.767} C_VEL
LIN {X 0,Y 580.291,Z 715.013,A -85,B 0,C 180,E1 -1838.146,E2 -1838.146} C_VEL
LIN {X 0,Y 580.302,Z 715.006,A -85,B 0,C 180,E1 -1840.843,E2 -1840.843} C_VEL
LIN {X 0,Y 580.281,Z 715.009,A -85,B 0,C 180,E1 -1843.658,E2 -1843.658} C_VEL
LIN {X 0,Y 580.278,Z 715.016,A -85,B 0,C 180,E1 -1846.609,E2 -1846.609} C_VEL
LIN {X 0,Y 580.303,Z 715.006,A -85,B 0,C 180,E1 -1849.157,E2 -1849.157} C_VEL
LIN {X 0,Y 580.292,Z 715.009,A -85,B 0,C 180,E1 -1851.927,E2 -1851.927} C_VEL
LIN {X 0,Y 580.309,Z 715.013,A -85,B 0,C 180,E1 -1854.457,E2 -1854.457} C_VEL
LIN {X 0,Y 580.293,Z 715.012,A -85,B 0,C 180,E1 -1856.975,E2 -1856.975} C_VEL
LIN {X 0,Y 580.303,Z 715.005,A -85,B 0,C 180,E1 -1859.425,E2 -1859.425} C_VEL
LIN {X 0,Y 580.299,Z 715.009,A -85,B 0,C 180,E1 -1862.141,E2 -1862.141} C_VEL
LIN {X 0,Y 580.323,Z 715.007,A -85,B 0,C 180,E1 -1865.27,E2 -1865.27} C_VEL
LIN {X 0,Y 580.325,Z 715.082,A -85,B 0,C 180,E1 -1868.37,E2 -1868.37} C_VEL
LIN {X 0,Y 580.651,Z 719.076,A -85,B 0,C 180,E1 -1869.106,E2 -1869.106} C_VEL
LIN {X 0,Y 580.524,Z 735.145,A -85,B 0,C 180,E1 -1871.836,E2 -1871.836} C_VEL
LIN {X 0,Y 580.39,Z 751.367,A -85,B 0,C 180,E1 -1874.55,E2 -1874.55} C_VEL
LIN {X 0,Y 580.276,Z 767.588,A -85,B 0,C 180,E1 -1877.23,E2 -1877.23} C_VEL
LIN {X 0,Y 580.239,Z 779.94,A -85,B 0,C 180,E1 -1879.223,E2 -1879.223} C_VEL
LIN {X 0,Y 580.554,Z 782.587,A -85,B 0,C 180,E1 -1879.299,E2 -1879.299} C_VEL
LIN {X 0,Y 580.592,Z 856.139,A -85,B 0,C 180,E1 -1880.221,E2 -1880.221} C_VEL
LIN {X 0,Y 580.513,Z 865.413,A -85,B 0,C 180,E1 -1880.418,E2 -1880.418} C_VEL
LIN {X 0,Y 580.456,Z 873.891,A -85,B 0,C 180,E1 -1880.68,E2 -1880.68} C_VEL
LIN {X 0,Y 580.421,Z 882.397,A -85,B 0,C 180,E1 -1881.031,E2 -1881.031} C_VEL
LIN {X 0,Y 580.362,Z 890.726,A -85,B 0,C 180,E1 -1881.469,E2 -1881.469} C_VEL
LIN {X 0,Y 580.31,Z 898.764,A -85,B 0,C 180,E1 -1881.994,E2 -1881.994} C_VEL
LIN {X 0,Y 580.24,Z 906.416,A -85,B 0,C 180,E1 -1882.606,E2 -1882.606} C_VEL
LIN {X 0,Y 580.217,Z 913.884,A -85,B 0,C 180,E1 -1883.335,E2 -1883.335} C_VEL
LIN {X 0,Y 580.173,Z 921.432,A -85,B 0,C 180,E1 -1884.264,E2 -1884.264} C_VEL
LIN {X 0,Y 580.084,Z 926.986,A -85,B 0,C 180,E1 -1885.135,E2 -1885.135} C_VEL
LIN {X 0,Y 580.137,Z 932.147,A -85,B 0,C 180,E1 -1886.18,E2 -1886.18} C_VEL
LIN {X 0,Y 580.07,Z 934.788,A -85,B 0,C 180,E1 -1886.875,E2 -1886.875} C_VEL
LIN {X 0,Y 580.037,Z 937.68,A -85,B 0,C 180,E1 -1887.917,E2 -1887.917} C_VEL
LIN {X 0,Y 580.045,Z 938.936,A -85,B 0,C 180,E1 -1888.611,E2 -1888.611} C_VEL
LIN {X 0,Y 580.038,Z 939.712,A -85,B 0,C 180,E1 -1889.306,E2 -1889.306} C_VEL
LIN {X 0,Y 580.034,Z 940,A -85,B 0,C 180,E1 -1890,E2 -1890} C_VEL
LIN {X 0,Y 580.038,Z 939.712,A -85,B 0,C 180,E1 -1890.694,E2 -1890.694} C_VEL
LIN {X 0,Y 580.045,Z 938.936,A -85,B 0,C 180,E1 -1891.389,E2 -1891.389} C_VEL
LIN {X 0,Y 580.037,Z 937.68,A -85,B 0,C 180,E1 -1892.083,E2 -1892.083} C_VEL
LIN {X 0,Y 580.07,Z 934.787,A -85,B 0,C 180,E1 -1893.125,E2 -1893.125} C_VEL
LIN {X 0,Y 580.137,Z 932.147,A -85,B 0,C 180,E1 -1893.82,E2 -1893.82} C_VEL
LIN {X 0,Y 580.084,Z 926.985,A -85,B 0,C 180,E1 -1894.865,E2 -1894.865} C_VEL
LIN {X 0,Y 580.173,Z 921.43,A -85,B 0,C 180,E1 -1895.736,E2 -1895.736} C_VEL
LIN {X 0,Y 580.209,Z 913.948,A -85,B 0,C 180,E1 -1896.659,E2 -1896.659} C_VEL
LIN {X 0,Y 580.24,Z 906.418,A -85,B 0,C 180,E1 -1897.394,E2 -1897.394} C_VEL
LIN {X 0,Y 580.31,Z 898.766,A -85,B 0,C 180,E1 -1898.006,E2 -1898.006} C_VEL
LIN {X 0,Y 580.362,Z 890.727,A -85,B 0,C 180,E1 -1898.531,E2 -1898.531} C_VEL
LIN {X 0,Y 580.421,Z 882.397,A -85,B 0,C 180,E1 -1898.969,E2 -1898.969} C_VEL
LIN {X 0,Y 580.456,Z 873.892,A -85,B 0,C 180,E1 -1899.32,E2 -1899.32} C_VEL
LIN {X 0,Y 580.537,Z 863.753,A -85,B 0,C 180,E1 -1899.626,E2 -1899.626} C_VEL
LIN {X 0,Y 580.586,Z 852.057,A -85,B 0,C 180,E1 -1899.845,E2 -1899.845} C_VEL
LIN {X 0,Y 580.536,Z 782.372,A -85,B 0,C 180,E1 -1900.704,E2 -1900.704} C_VEL
LIN {X 0,Y 580.238,Z 779.936,A -85,B 0,C 180,E1 -1900.777,E2 -1900.777} C_VEL
LIN {X 0,Y 580.33,Z 763.263,A -85,B 0,C 180,E1 -1903.481,E2 -1903.481} C_VEL
LIN {X 0,Y 580.48,Z 744.878,A -85,B 0,C 180,E1 -1906.53,E2 -1906.53} C_VEL
LIN {X 0,Y 580.613,Z 726.437,A -85,B 0,C 180,E1 -1909.637,E2 -1909.637} C_VEL
LIN {X 0,Y 580.59,Z 716.761,A -85,B 0,C 180,E1 -1911.294,E2 -1911.294} C_VEL
LIN {X 0,Y 580.329,Z 715.038,A -85,B 0,C 180,E1 -1911.653,E2 -1911.653} C_VEL
LIN {X 0,Y 580.323,Z 715.007,A -85,B 0,C 180,E1 -1914.73,E2 -1914.73} C_VEL
LIN {X 0,Y 580.299,Z 715.009,A -85,B 0,C 180,E1 -1917.859,E2 -1917.859} C_VEL
LIN {X 0,Y 580.293,Z 715.007,A -85,B 0,C 180,E1 -1920.696,E2 -1920.696} C_VEL
LIN {X 0,Y 580.306,Z 715.016,A -85,B 0,C 180,E1 -1923.317,E2 -1923.317} C_VEL
LIN {X 0,Y 580.328,Z 715.007,A -85,B 0,C 180,E1 -1925.768,E2 -1925.768} C_VEL
LIN {X 0,Y 580.291,Z 715.009,A -85,B 0,C 180,E1 -1928.146,E2 -1928.146} C_VEL
LIN {X 0,Y 580.302,Z 715.006,A -85,B 0,C 180,E1 -1930.843,E2 -1930.843} C_VEL
LIN {X 0,Y 580.28,Z 715.018,A -85,B 0,C 180,E1 -1933.658,E2 -1933.658} C_VEL
LIN {X 0,Y 580.28,Z 715.008,A -85,B 0,C 180,E1 -1936.609,E2 -1936.609} C_VEL
LIN {X 0,Y 580.302,Z 715.006,A -85,B 0,C 180,E1 -1939.157,E2 -1939.157} C_VEL
LIN {X 0,Y 580.293,Z 715.012,A -85,B 0,C 180,E1 -1941.927,E2 -1941.927} C_VEL
LIN {X 0,Y 580.309,Z 715.006,A -85,B 0,C 180,E1 -1944.457,E2 -1944.457} C_VEL
LIN {X 0,Y 580.293,Z 715.007,A -85,B 0,C 180,E1 -1946.975,E2 -1946.975} C_VEL
LIN {X 0,Y 580.305,Z 715.008,A -85,B 0,C 180,E1 -1949.426,E2 -1949.426} C_VEL
LIN {X 0,Y 580.301,Z 715.013,A -85,B 0,C 180,E1 -1952.141,E2 -1952.141} C_VEL
LIN {X 0,Y 580.323,Z 715.004,A -85,B 0,C 180,E1 -1955.27,E2 -1955.27} C_VEL
LIN {X 0,Y 580.275,Z 715.017,A -85,B 0,C 180,E1 -1957.948,E2 -1957.948} C_VEL
LIN {X 0,Y 580.322,Z 715.004,A -85,B 0,C 180,E1 -1960.914,E2 -1960.914} C_VEL
LIN {X 0,Y 580.283,Z 715.013,A -85,B 0,C 180,E1 -1963.826,E2 -1963.826} C_VEL
LIN {X 0,Y 580.328,Z 715.009,A -85,B 0,C 180,E1 -1965.983,E2 -1965.983} C_VEL
LIN {X 0,Y 580.307,Z 715.006,A -85,B 0,C 180,E1 -1968.827,E2 -1968.827} C_VEL
LIN {X 0,Y 580.336,Z 715.003,A -85,B 0,C 180,E1 -1971.644,E2 -1971.644} C_VEL
LIN {X 0,Y 580.32,Z 715.013,A -85,B 0,C 180,E1 -1974.44,E2 -1974.44} C_VEL
LIN {X 0,Y 580.346,Z 714.998,A -85,B 0,C 180,E1 -1977.224,E2 -1977.224} C_VEL
LIN {X 0,Y 580.355,Z 715.001,A -85,B 0,C 180,E1 -1980,E2 -1980} C_VEL
LIN {X 0,Y 580.345,Z 715.008,A -85,B 0,C 180,E1 -1982.777,E2 -1982.777} C_VEL
LIN {X 0,Y 580.328,Z 715.002,A -85,B 0,C 180,E1 -1985.56,E2 -1985.56} C_VEL
LIN {X 0,Y 580.332,Z 715.004,A -85,B 0,C 180,E1 -1988.356,E2 -1988.356} C_VEL
LIN {X 0,Y 580.303,Z 715.009,A -85,B 0,C 180,E1 -1991.191,E2 -1991.191} C_VEL
LIN {X 0,Y 580.328,Z 715.003,A -85,B 0,C 180,E1 -1994.017,E2 -1994.017} C_VEL
LIN {X 0,Y 580.315,Z 715.012,A -85,B 0,C 180,E1 -1996.914,E2 -1996.914} C_VEL
LIN {X 0,Y 580.29,Z 715.007,A -85,B 0,C 180,E1 -1999.823,E2 -1999.823} C_VEL
LIN {X 0,Y 580.285,Z 715.013,A -85,B 0,C 180,E1 -2001.329,E2 -2001.329} C_VEL
LIN {X 0,Y 579.587,Z 715.098,A -85,B 0,C 180,E1 -2001.908,E2 -2001.908} C_VEL
LIN {X 0,Y 576.708,Z 715.462,A -85,B 0,C 180,E1 -2002.848,E2 -2002.848} C_VEL
LIN {X 0,Y 574.313,Z 715.755,A -85,B 0,C 180,E1 -2003.604,E2 -2003.604} C_VEL
LIN {X 0,Y 573.315,Z 715.876,A -85,B 0,C 180,E1 -2004.188,E2 -2004.188} C_VEL
LIN {X 0,Y 573.249,Z 715.885,A -85,B 0,C 180,E1 -2004.385,E2 -2004.385} C_VEL
LIN {X 0,Y 573.253,Z 715.891,A -85,B 0,C 180,E1 -2006.976,E2 -2006.976} C_VEL
LIN {X 0,Y 573.242,Z 715.89,A -85,B 0,C 180,E1 -2009.487,E2 -2009.487} C_VEL
LIN {X 0,Y 573.256,Z 715.885,A -85,B 0,C 180,E1 -2012.645,E2 -2012.645} C_VEL
LIN {X 0,Y 573.209,Z 715.899,A -85,B 0,C 180,E1 -2015.188,E2 -2015.188} C_VEL
LIN {X 0,Y 573.233,Z 715.889,A -85,B 0,C 180,E1 -2017.808,E2 -2017.808} C_VEL
LIN {X 0,Y 573.246,Z 715.883,A -85,B 0,C 180,E1 -2020.525,E2 -2020.525} C_VEL
LIN {X 0,Y 573.238,Z 715.889,A -85,B 0,C 180,E1 -2023.359,E2 -2023.359} C_VEL
LIN {X 0,Y 573.239,Z 715.886,A -85,B 0,C 180,E1 -2026.641,E2 -2026.641} C_VEL
LIN {X 0,Y 573.246,Z 715.895,A -85,B 0,C 180,E1 -2029.475,E2 -2029.475} C_VEL
LIN {X 0,Y 573.235,Z 715.886,A -85,B 0,C 180,E1 -2032.192,E2 -2032.192} C_VEL
LIN {X 0,Y 573.235,Z 715.891,A -85,B 0,C 180,E1 -2035.229,E2 -2035.229} C_VEL
LIN {X 0,Y 573.239,Z 715.887,A -85,B 0,C 180,E1 -2038.184,E2 -2038.184} C_VEL
LIN {X 0,Y 573.259,Z 715.884,A -85,B 0,C 180,E1 -2040.634,E2 -2040.634} C_VEL
LIN {X 0,Y 573.225,Z 715.893,A -85,B 0,C 180,E1 -2043.51,E2 -2043.51} C_VEL
LIN {X 0,Y 573.226,Z 715.893,A -85,B 0,C 180,E1 -2046.134,E2 -2046.134} C_VEL
LIN {X 0,Y 573.251,Z 715.886,A -85,B 0,C 180,E1 -2049.174,E2 -2049.174} C_VEL
LIN {X 0,Y 573.268,Z 715.982,A -85,B 0,C 180,E1 -2051.783,E2 -2051.783} C_VEL
LIN {X 0,Y 573.283,Z 724.597,A -85,B 0,C 180,E1 -2053.623,E2 -2053.623} C_VEL
LIN {X 0,Y 573.188,Z 738.523,A -85,B 0,C 180,E1 -2056.528,E2 -2056.528} C_VEL
LIN {X 0,Y 573.135,Z 751.293,A -85,B 0,C 180,E1 -2059.13,E2 -2059.13} C_VEL
LIN {X 0,Y 573.315,Z 753.129,A -85,B 0,C 180,E1 -2059.211,E2 -2059.211} C_VEL
LIN {X 0,Y 573.644,Z 761.581,A -85,B 0,C 180,E1 -2059.326,E2 -2059.326} C_VEL
LIN {X 0,Y 573.557,Z 827.42,A -85,B 0,C 180,E1 -2060.167,E2 -2060.167} C_VEL
LIN {X 0,Y 573.509,Z 837.897,A -85,B 0,C 180,E1 -2060.411,E2 -2060.411} C_VEL
LIN {X 0,Y 573.433,Z 849.581,A -85,B 0,C 180,E1 -2060.832,E2 -2060.832} C_VEL
LIN {X 0,Y 573.343,Z 859.977,A -85,B 0,C 180,E1 -2061.364,E2 -2061.364} C_VEL
LIN {X 0,Y 573.257,Z 868.153,A -85,B 0,C 180,E1 -2061.895,E2 -2061.895} C_VEL
LIN {X 0,Y 573.191,Z 875.905,A -85,B 0,C 180,E1 -2062.515,E2 -2062.515} C_VEL
LIN {X 0,Y 573.156,Z 884.137,A -85,B 0,C 180,E1 -2063.323,E2 -2063.323} C_VEL
LIN {X 0,Y 573.113,Z 891.131,A -85,B 0,C 180,E1 -2064.194,E2 -2064.194} C_VEL
LIN {X 0,Y 573.004,Z 896.742,A -85,B 0,C 180,E1 -2065.075,E2 -2065.075} C_VEL
LIN {X 0,Y 573.036,Z 901.955,A -85,B 0,C 180,E1 -2066.132,E2 -2066.132} C_VEL
LIN {X 0,Y 572.992,Z 904.643,A -85,B 0,C 180,E1 -2066.836,E2 -2066.836} C_VEL
LIN {X 0,Y 572.94,Z 907.58,A -85,B 0,C 180,E1 -2067.891,E2 -2067.891} C_VEL
LIN {X 0,Y 572.944,Z 908.875,A -85,B 0,C 180,E1 -2068.594,E2 -2068.594} C_VEL
LIN {X 0,Y 572.936,Z 909.691,A -85,B 0,C 180,E1 -2069.297,E2 -2069.297} C_VEL
LIN {X 0,Y 572.936,Z 909.996,A -85,B 0,C 180,E1 -2070,E2 -2070} C_VEL
LIN {X 0,Y 572.937,Z 909.732,A -85,B 0,C 180,E1 -2070.703,E2 -2070.703} C_VEL
LIN {X 0,Y 572.945,Z 908.997,A -85,B 0,C 180,E1 -2071.406,E2 -2071.406} C_VEL
LIN {X 0,Y 572.941,Z 907.784,A -85,B 0,C 180,E1 -2072.109,E2 -2072.109} C_VEL
LIN {X 0,Y 572.991,Z 904.936,A -85,B 0,C 180,E1 -2073.164,E2 -2073.164} C_VEL
LIN {X 0,Y 573.025,Z 902.342,A -85,B 0,C 180,E1 -2073.868,E2 -2073.868} C_VEL
LIN {X 0,Y 572.983,Z 897.231,A -85,B 0,C 180,E1 -2074.925,E2 -2074.925} C_VEL
LIN {X 0,Y 573.113,Z 891.731,A -85,B 0,C 180,E1 -2075.806,E2 -2075.806} C_VEL
LIN {X 0,Y 573.156,Z 883.341,A -85,B 0,C 180,E1 -2076.849,E2 -2076.849} C_VEL
LIN {X 0,Y 573.215,Z 875.922,A -85,B 0,C 180,E1 -2077.574,E2 -2077.574} C_VEL
LIN {X 0,Y 573.284,Z 868.171,A -85,B 0,C 180,E1 -2078.193,E2 -2078.193} C_VEL
LIN {X 0,Y 573.356,Z 859.997,A -85,B 0,C 180,E1 -2078.725,E2 -2078.725} C_VEL
LIN {X 0,Y 573.433,Z 849.604,A -85,B 0,C 180,E1 -2079.257,E2 -2079.257} C_VEL
LIN {X 0,Y 573.522,Z 837.934,A -85,B 0,C 180,E1 -2079.678,E2 -2079.678} C_VEL
LIN {X 0,Y 573.597,Z 827.474,A -85,B 0,C 180,E1 -2079.922,E2 -2079.922} C_VEL
LIN {X 0,Y 573.647,Z 756.77,A -85,B 0,C 180,E1 -2080.824,E2 -2080.824} C_VEL
LIN {X 0,Y 573.163,Z 751.854,A -85,B 0,C 180,E1 -2080.912,E2 -2080.912} C_VEL
LIN {X 0,Y 573.148,Z 750.703,A -85,B 0,C 180,E1 -2081.048,E2 -2081.048} C_VEL
LIN {X 0,Y 573.193,Z 737.216,A -85,B 0,C 180,E1 -2083.833,E2 -2083.833} C_VEL
LIN {X 0,Y 573.306,Z 723.485,A -85,B 0,C 180,E1 -2086.7,E2 -2086.7} C_VEL
LIN {X 0,Y 573.321,Z 715.985,A -85,B 0,C 180,E1 -2088.308,E2 -2088.308} C_VEL
LIN {X 0,Y 573.253,Z 715.885,A -85,B 0,C 180,E1 -2091.291,E2 -2091.291} C_VEL
LIN {X 0,Y 573.221,Z 715.893,A -85,B 0,C 180,E1 -2093.866,E2 -2093.866} C_VEL
LIN {X 0,Y 573.203,Z 715.898,A -85,B 0,C 180,E1 -2096.485,E2 -2096.485} C_VEL
LIN {X 0,Y 573.258,Z 715.884,A -85,B 0,C 180,E1 -2099.366,E2 -2099.366} C_VEL
LIN {X 0,Y 573.251,Z 715.891,A -85,B 0,C 180,E1 -2102.228,E2 -2102.228} C_VEL
LIN {X 0,Y 573.206,Z 715.891,A -85,B 0,C 180,E1 -2105.188,E2 -2105.188} C_VEL
LIN {X 0,Y 573.234,Z 715.886,A -85,B 0,C 180,E1 -2107.808,E2 -2107.808} C_VEL
LIN {X 0,Y 573.246,Z 715.894,A -85,B 0,C 180,E1 -2110.525,E2 -2110.525} C_VEL
LIN {X 0,Y 573.238,Z 715.887,A -85,B 0,C 180,E1 -2113.359,E2 -2113.359} C_VEL
LIN {X 0,Y 573.238,Z 715.891,A -85,B 0,C 180,E1 -2116.641,E2 -2116.641} C_VEL
LIN {X 0,Y 573.246,Z 715.883,A -85,B 0,C 180,E1 -2119.475,E2 -2119.475} C_VEL
LIN {X 0,Y 573.233,Z 715.888,A -85,B 0,C 180,E1 -2122.192,E2 -2122.192} C_VEL
LIN {X 0,Y 573.236,Z 715.889,A -85,B 0,C 180,E1 -2125.229,E2 -2125.229} C_VEL
LIN {X 0,Y 573.241,Z 715.885,A -85,B 0,C 180,E1 -2128.184,E2 -2128.184} C_VEL
LIN {X 0,Y 573.26,Z 715.889,A -85,B 0,C 180,E1 -2130.634,E2 -2130.634} C_VEL
LIN {X 0,Y 573.236,Z 715.886,A -85,B 0,C 180,E1 -2133.508,E2 -2133.508} C_VEL
LIN {X 0,Y 573.229,Z 715.886,A -85,B 0,C 180,E1 -2136.134,E2 -2136.134} C_VEL
LIN {X 0,Y 573.253,Z 715.894,A -85,B 0,C 180,E1 -2139.174,E2 -2139.174} C_VEL
LIN {X 0,Y 573.223,Z 715.892,A -85,B 0,C 180,E1 -2141.411,E2 -2141.411} C_VEL
LIN {X 0,Y 573.253,Z 715.886,A -85,B 0,C 180,E1 -2143.622,E2 -2143.622} C_VEL
LIN {X 0,Y 573.275,Z 715.883,A -85,B 0,C 180,E1 -2145.807,E2 -2145.807} C_VEL
LIN {X 0,Y 573.266,Z 715.885,A -85,B 0,C 180,E1 -2148.745,E2 -2148.745} C_VEL
LIN {X 0,Y 573.288,Z 715.884,A -85,B 0,C 180,E1 -2151.54,E2 -2151.54} C_VEL
LIN {X 0,Y 573.295,Z 715.877,A -85,B 0,C 180,E1 -2154.372,E2 -2154.372} C_VEL
LIN {X 0,Y 573.316,Z 715.88,A -85,B 0,C 180,E1 -2157.892,E2 -2157.892} C_VEL
LIN {X 0,Y 573.335,Z 715.873,A -85,B 0,C 180,E1 -2160.702,E2 -2160.702} C_VEL
LIN {X 0,Y 573.234,Z 715.892,A -85,B 0,C 180,E1 -2163.514,E2 -2163.514} C_VEL
LIN {X 0,Y 573.287,Z 715.89,A -85,B 0,C 180,E1 -2165.628,E2 -2165.628} C_VEL
LIN {X 0,Y 573.292,Z 715.88,A -85,B 0,C 180,E1 -2168.459,E2 -2168.459} C_VEL
LIN {X 0,Y 573.274,Z 715.883,A -85,B 0,C 180,E1 -2171.312,E2 -2171.312} C_VEL
LIN {X 0,Y 573.284,Z 715.881,A -85,B 0,C 180,E1 -2174.424,E2 -2174.424} C_VEL
LIN {X 0,Y 573.262,Z 715.884,A -85,B 0,C 180,E1 -2177.111,E2 -2177.111} C_VEL
LIN {X 0,Y 573.255,Z 715.889,A -85,B 0,C 180,E1 -2180.076,E2 -2180.076} C_VEL
LIN {X 0,Y 573.236,Z 715.885,A -85,B 0,C 180,E1 -2183.099,E2 -2183.099} C_VEL
LIN {X 0,Y 573.256,Z 715.885,A -85,B 0,C 180,E1 -2185.41,E2 -2185.41} C_VEL
LIN {X 0,Y 573.266,Z 715.892,A -85,B 0,C 180,E1 -2188.031,E2 -2188.031} C_VEL
LIN {X 0,Y 573.24,Z 715.886,A -85,B 0,C 180,E1 -2190.884,E2 -2190.884} C_VEL
LIN {X 0,Y 573.264,Z 715.884,A -85,B 0,C 180,E1 -2193.524,E2 -2193.524} C_VEL
LIN {X 0,Y 573.263,Z 715.889,A -85,B 0,C 180,E1 -2196.048,E2 -2196.048} C_VEL
LIN {X 0,Y 573.251,Z 715.881,A -85,B 0,C 180,E1 -2198.701,E2 -2198.701} C_VEL
LIN {X 0,Y 573.255,Z 715.882,A -85,B 0,C 180,E1 -2201.596,E2 -2201.596} C_VEL
LIN {X 0,Y 573.237,Z 715.896,A -85,B 0,C 180,E1 -2204.333,E2 -2204.333} C_VEL
LIN {X 0,Y 573.242,Z 715.884,A -85,B 0,C 180,E1 -2207.358,E2 -2207.358} C_VEL
LIN {X 0,Y 573.25,Z 715.892,A -85,B 0,C 180,E1 -2210.393,E2 -2210.393} C_VEL
LIN {X 0,Y 573.257,Z 715.885,A -85,B 0,C 180,E1 -2213.078,E2 -2213.078} C_VEL
LIN {X 0,Y 573.276,Z 715.882,A -85,B 0,C 180,E1 -2215.672,E2 -2215.672} C_VEL
LIN {X 0,Y 573.25,Z 715.887,A -85,B 0,C 180,E1 -2218.185,E2 -2218.185} C_VEL
LIN {X 0,Y 573.267,Z 715.889,A -85,B 0,C 180,E1 -2220.634,E2 -2220.634} C_VEL
LIN {X 0,Y 573.239,Z 715.887,A -85,B 0,C 180,E1 -2223.507,E2 -2223.507} C_VEL
LIN {X 0,Y 573.233,Z 715.887,A -85,B 0,C 180,E1 -2226.135,E2 -2226.135} C_VEL
LIN {X 0,Y 573.325,Z 716.052,A -85,B 0,C 180,E1 -2228.281,E2 -2228.281} C_VEL
LIN {X 0,Y 573.693,Z 721.087,A -85,B 0,C 180,E1 -2229.19,E2 -2229.19} C_VEL
LIN {X 0,Y 573.523,Z 738.39,A -85,B 0,C 180,E1 -2232.16,E2 -2232.16} C_VEL
LIN {X 0,Y 573.374,Z 755.693,A -85,B 0,C 180,E1 -2235.084,E2 -2235.084} C_VEL
LIN {X 0,Y 573.232,Z 774.077,A -85,B 0,C 180,E1 -2238.149,E2 -2238.149} C_VEL
LIN {X 0,Y 573.174,Z 780.009,A -85,B 0,C 180,E1 -2239.093,E2 -2239.093} C_VEL
LIN {X 0,Y 573.536,Z 782.904,A -85,B 0,C 180,E1 -2239.17,E2 -2239.17} C_VEL
LIN {X 0,Y 573.603,Z 856.138,A -85,B 0,C 180,E1 -2240.101,E2 -2240.101} C_VEL
LIN {X 0,Y 573.523,Z 865.413,A -85,B 0,C 180,E1 -2240.3,E2 -2240.3} C_VEL
LIN {X 0,Y 573.455,Z 873.892,A -85,B 0,C 180,E1 -2240.566,E2 -2240.566} C_VEL
LIN {X 0,Y 573.413,Z 882.399,A -85,B 0,C 180,E1 -2240.921,E2 -2240.921} C_VEL
LIN {X 0,Y 573.341,Z 890.728,A -85,B 0,C 180,E1 -2241.364,E2 -2241.364} C_VEL
LIN {X 0,Y 573.26,Z 898.766,A -85,B 0,C 180,E1 -2241.895,E2 -2241.895} C_VEL
LIN {X 0,Y 573.19,Z 906.416,A -85,B 0,C 180,E1 -2242.514,E2 -2242.514} C_VEL
LIN {X 0,Y 573.151,Z 914.582,A -85,B 0,C 180,E1 -2243.326,E2 -2243.326} C_VEL
LIN {X 0,Y 573.112,Z 921.433,A -85,B 0,C 180,E1 -2244.194,E2 -2244.194} C_VEL
LIN {X 0,Y 572.995,Z 926.987,A -85,B 0,C 180,E1 -2245.075,E2 -2245.075} C_VEL
LIN {X 0,Y 573.036,Z 932.148,A -85,B 0,C 180,E1 -2246.132,E2 -2246.132} C_VEL
